	RAMP4:RAMP_INT;
	RAMP5:RAMP_INT;
	RAMP6:RAMP_INT;
	RAMP7:RAMP_INT;
	RAMP8:RAMP_INT;
	RAMP9:RAMP_INT;
	RAMP10:RAMP_INT;
	RAMP11:RAMP_INT;
	RAMP12:RAMP_INT;
	RAMP13:RAMP_INT;
	RAMP14:RAMP_INT;
	RAMP15:RAMP_INT;
	RAMP16:RAMP_INT;
	RAMP17:RAMP_INT;
	RAMP18:RAMP_INT;
	RAMP19:RAMP_INT;
	RAMP20:RAMP_INT;
	RAMP21:RAMP_INT;
	RAMP22:RAMP_INT;
	RAMP23:RAMP_INT;
	RAMP24:RAMP_INT;
	PWM_Y23_SET_Taget1:INT;
	PWM_Y24_SET_Taget1:INT;
	PWM_Y18_SET_Taget1:INT;
	PWM_Y18_SET_Taget:UINT;
	ASCEND_value2:INT;
	//2023 01 13 增加
	//行走动作斜坡值
	R_RAMP_traval:INT:=800;
	F_RAMP_traval:INT:=400;
	TIMEBASE_traval:TIME:=T#200MS;
	//动力头动作斜坡值
	R_RAMP_ratate:INT:=800;
	F_RAMP_ratate:INT:=800;
	TIMEBASE_ratate:TIME:=T#100MS;
	//主卷扬动作斜坡值
	R_RAMP_mainwinch:INT:=800;
	F_RAMP_mainwinch_up:INT:=400;
	F_RAMP_mainwinch_down:INT:=400;
	TIMEBASE_mainwinch:TIME:=T#200MS;
	//主泵排量斜坡值
	R_RAMP_pump:INT:=300;
	F_RAMP_pump:INT:=1000;
	TIMEBASE_pump:TIME:=T#1000MS;
	//卸荷阀斜坡值
	R_RAMP_xiehe:INT:=500;
	F_RAMP_xiehe:INT:=400;
	TIMEBASE_xiehe:TIME:=T#500MS;
	
	//直线阀斜坡值
	R_RAMP_zhixian:INT:=800;
	F_RAMP_zhixian:INT:=800;
	TIMEBASE_zhixian:TIME:=T#300MS;
		
	Subtract: BOOL;
	TIME_LvBo4:TON;
	Curve_input:UINT;
	Curve_Par: SINT:=0;
	Curve_Par1: SINT:=0;
	Move_JOY_FUHE: UINT;
	PWM_JOY_Jiao_L_UP1:UINT;
	PWM_JOY_Jiao_L_DOWN1:UINT;
	PWM_JOY_Jiao_R_UP1:UINT;
	PWM_JOY_Jiao_R_DOWN1:UINT;
	
	PWM_JOYX_R_UP_a:UINT;
	PWM_JOYX_R_UP_b:UINT;
	
	PWM_JOYX_R_DOWN_a:UINT;
	PWM_JOYX_R_DOWN_b:UINT;
	
	PWM_JOYY_L_DOWN_a:UINT;
	PWM_JOYY_L_DOWN_b:UINT;
	
	PWM_JOYY_L_UP_a:UINT;
	PWM_JOYY_L_UP_b:UINT;
	aaaa:UINT:=500;
	
	JOY_PAOTU:BOOL;
	
	JOY_PAOTU_tiaojian:BOOL;
	TIME_1000_1ms:ton;
	tempbool:BOOL;
	CANI_JOYX_R_last2:UINT;
	Sub_Joyx_r2:INT;
	JianGE11:REAL:=2;
	JianGE21:uint:=10;
	END_IFc: INT;
	x1:UINT:=8;
	x2:UINT:=8;
	PWM_JOY_JIAO:UINT;
	PWM_Y39_SET1:UINT;
	PWM_Y40_SET1:UINT;
	aaa: INT;
	TIME_50ms:TON;
	TIME_55ms:TOF;
	TIME_2000ms:TOF;
	start_move: BOOL;
	T1:TIME;
	TEMP1:UINT;
	X3: INT;
	X4: INT;
	liandong:BOOL;
	PWM_Y9_SET1:INT;
	PWM_Y10_SET1:INT;
	PWM_Y13_SET1:INT;
	PWM_Y14_SET1:INT;
	yanchi1:BOOL;
	yanchi_ton1:ton;
	RAMP15_IN:UINT;
	RAMP16_IN:UINT;
	Rtrig_d1:R_TRIG;
	Rtrig_d2:R_TRIG;
	
	Rtrig_DongLiTou1:R_TRIG;
	Rtrig_DongLiTou2:R_TRIG;
	Count_TIMES_Fanzhuan: UINT;
	Count_TIMES_Zhengzhuan: UINT;
	TIME_1000ms:TON;
	TIME_1000ms_TP:TON;
	Count_TIMES_Fanzhuan_LAST: UINT;
	Count_TIMES_Zhengzhuan_LAST: UINT;
	Paotu_Modle: BOOL;
	PaoTU_biaozhi: BOOL;
	TIMEBASE_D: TIME;
	PWM_Y39_SET_Target1:INT;
	PWM_Y40_SET_Target1:INT;
	PWM_Y37_SET_Target:UINT;
	PWM_Y17_SET2:UINT;
	t_PowerHead_move:TON;
	x_t_PowerHead_move:INT:=10;//100-10
	x2_t_PowerHead_move:INT:=10;//100-10
	P_value:REAL;//动力头反转+主卷上提时的分流系数
	PWM_JOY_P:UINT;
	PWM_JOY_P1:UINT;
	PWM_JOY_P2:UINT;
	PWM_JOY_P3:UINT;
	PWM_JOY_P4:UINT;
	ASCEND_value:INT;
	ftp1:INT:=500;
	ftp2:INT:=100;
	t_powertime:TIME;
	
	P25_Flag:BOOL;
	P27_Flag:BOOL;
	P29_Flag:BOOL;
	P31_Flag:BOOL;
	PressLvBo_TON:TON;
	PressLvBo_TON1: TON;
	PressLvBo_TON2: TON;
	PressLvBo_TON3: TON;
	test: BYTE;
	testpaotu: UINT := 450;
	Y33_2:UINT:=370;
	Y33_1:UINT:=200;
END_VAR

//动力头反转与主卷上提时的分流系数值
(*IF CANO_ZhuJuanPressure<=100 THEN
	P_value:=TO_REAL(PAR_KI+40)/100.0;
ELSIF CANO_ZhuJuanPressure>100 AND  CANO_ZhuJuanPressure<=200 THEN
	P_value:=TO_REAL(PAR_KI+20)/100.0;
ELSE
	P_value:=TO_REAL(PAR_KI)/100;
END_IF*)
P_value:=TO_REAL(PAR_KI)/100;  //出厂值设定为35
//喇叭
IF DI_LHandle_SB5 THEN
	DOH_Y59:=TRUE;
ELSE
	DOH_Y59:=FALSE;
END_IF
//延时断电
TIME_2000ms(IN:=DIH_power3,PT:=T#2S);
IF(TIME_2000ms.Q)THEN
	DOH_YS3:=TRUE;
ELSE
	DOH_YS3:=FALSE;
END_IF

//主卷上限位及解锁
IF(DI_LHandle_SB1 AND (NOT CANI_WorkModeSwitch))THEN
	JieSuoBool:=TRUE;
ELSE
	JieSuoBool:=FALSE;	
END_IF

IF DIL_SQ4 THEN
	IF(NOT JieSuoBool) THEN
		PWM_JOYY_L_DOWN:=0;
	END_IF
END_IF

//主卷下限位及解锁
//主卷下放限制
IF( CANO_MainWinchTension*100<PAR_MainWinchLaLi_Low) AND (NOT DI_LHandle_SB1) AND (CANI_WorkModeSwitch)THEN
	PWM_JOYY_L_UP:=0;
END_IF

TIME_50ms(in:=start_move,pt:=T1);
TIME_55ms(in:=start_move,pt:=T#500MS);
IF( LeftMove_move OR  RightMove_move  OR   MainWinch_move OR PowerHead_move OR ViceWinch_move )THEN
	start_move:=TRUE;
ELSE
	start_move:=FALSE;
END_IF
	 


IF NOT DIL_SQ3 THEN(*先导控制输入*)
	IF PWM_JOYX_L_UP>10 OR PWM_JOYX_L_DOWN>10 THEN  DI_PWM_JOYX_L := TRUE;ELSE DI_PWM_JOYX_L:=FALSE;END_IF(*左手柄左右动作*)
	IF PWM_JOYY_L_UP>10 OR PWM_JOYY_L_DOWN>10 THEN  DI_PWM_JOYY_L := TRUE;ELSE DI_PWM_JOYY_L:=FALSE;END_IF(*左手柄前后动作*)
	IF PWM_JOYX_R_UP>10 OR PWM_JOYX_R_DOWN>10 THEN  DI_PWM_JOYX_R := TRUE;ELSE DI_PWM_JOYX_R:=FALSE;END_IF(*右手柄左右动作*)
	IF PWM_JOYY_R_UP>10 OR PWM_JOYY_R_DOWN>10 THEN  DI_PWM_JOYY_R := TRUE;ELSE DI_PWM_JOYY_R:=FALSE;END_IF(*右手柄前后动作*)
	IF PWM_JOY_Jiao_L_UP>10 OR PWM_JOY_Jiao_L_DOWN>10 THEN  DI_PWM_JOY_Jiao_L:= TRUE;ELSE DI_PWM_JOY_Jiao_L:=FALSE;END_IF(*左脚踏前后动作*)
	IF PWM_JOY_Jiao_R_UP>10 OR PWM_JOY_Jiao_R_DOWN>10 THEN  DI_PWM_JOY_Jiao_R := TRUE;ELSE DI_PWM_JOY_Jiao_R:=FALSE;END_IF(*左脚踏左右动作*)
ELSE
	DI_PWM_JOYX_L:=FALSE;
	DI_PWM_JOYY_L:=FALSE;
	DI_PWM_JOYX_R:=FALSE;
	DI_PWM_JOYY_R:=FALSE;
	DI_PWM_JOY_Jiao_L:=FALSE;
	DI_PWM_JOY_Jiao_R:=FALSE;
END_IF

(*动作标志*)
IF DI_PWM_JOYY_L THEN MainWinch_move:=TRUE; ELSE MainWinch_move:=FALSE;END_IF(*主卷扬动作*)
IF DI_PWM_JOYX_L THEN Rotation_move:=TRUE; ELSE Rotation_move:=FALSE;END_IF(*回转动作*)
IF CANI_WorkModeSwitch THEN   (*作业挡情况下*)
	IF DI_PWM_JOYX_R THEN PowerHead_move:=TRUE;ELSE PowerHead_move:=FALSE;END_IF(*动力头回转动作*)
	IF DI_PWM_JOYY_R THEN JiaYa_move:=TRUE;ELSE JiaYa_move:=FALSE;END_IF(*动力头加压动作*)
	LvZhang_move:=FALSE;
	BianFu_move:=FALSE;
	ViceWinch_move:=FALSE;
	LeftMove_move:=FALSE;
	RightMove_move:=FALSE;
ELSE   (*调整档状态*)
	IF DI_PWM_JOYX_R THEN  LvZhang_move:=TRUE;ELSE LvZhang_move:=FALSE;END_IF(*L履带、张紧、支腿动作,M4阀*)
	(*LeftMove_move:=DI_PWM_JOY_Jiao_L;(*左行走动作*)
	RightMove_move:=DI_PWM_JOY_Jiao_R;*)(*右行走动作*)
	IF( PWM_JOY_Jiao_L_UP1>10 OR PWM_JOY_Jiao_L_DOWN1>10)  AND  DI_PWM_JOY_Jiao_L THEN
		LeftMove_move:=TRUE;
	ELSE
		LeftMove_move:=FALSE;
	END_IF
	IF( PWM_JOY_Jiao_R_UP1>10 OR PWM_JOY_Jiao_R_DOWN1>10)  AND  DI_PWM_JOY_Jiao_R THEN
		RightMove_move:=TRUE;
	ELSE
		RightMove_move:=FALSE;
	END_IF

	IF  DI_RHandle_SB5 THEN
		ViceWinch_move:=FALSE;
		IF  DI_PWM_JOYY_R  THEN BianFu_move:=TRUE;ELSE BianFu_move:=FALSE;END_IF(*变幅动作M4阀*)
	ELSE
		BianFu_move:=FALSE;
		IF DI_PWM_JOYY_R  THEN ViceWinch_move:=TRUE;ELSE ViceWinch_move:=FALSE;END_IF(*副卷扬动作M4阀*)
	END_IF
	PowerHead_move:=FALSE;
	JiaYa_move:=FALSE;
END_IF


(****主阀单动作标志****)
	IF (NOT MainWinch_move) AND (NOT PowerHead_move) AND (ViceWinch_move) THEN
		Single_move:=TRUE;
	ELSE
		Single_move:=FALSE;
	END_IF
	
//先导控制
IF(NOT DIL_SQ3) AND NOT VarGpsSystemLockedState THEN
	DOH_Y51:=TRUE;
ELSE
	DOH_Y51:=FALSE;
END_IF

//行走动作
(*脚踏阀偏差*)
IF   ((PWM_JOY_Jiao_L_UP-PWM_JOY_Jiao_R_UP)<200 OR(PWM_JOY_Jiao_R_UP-PWM_JOY_Jiao_L_UP)<200) THEN
	PWM_JOY_Jiao_L_UP1:=MAX(PWM_JOY_Jiao_L_UP,PWM_JOY_Jiao_R_UP);
	PWM_JOY_Jiao_R_UP1:=MAX(PWM_JOY_Jiao_L_UP,PWM_JOY_Jiao_R_UP);
ELSE
	PWM_JOY_Jiao_L_UP1:=PWM_JOY_Jiao_L_UP;
	PWM_JOY_Jiao_R_UP1:=PWM_JOY_Jiao_R_UP;
END_IF
IF   ((PWM_JOY_Jiao_L_DOWN-PWM_JOY_Jiao_R_DOWN)<200  OR  (PWM_JOY_Jiao_R_DOWN-PWM_JOY_Jiao_L_DOWN)<200 ) THEN
	PWM_JOY_Jiao_L_DOWN1:=MAX(PWM_JOY_Jiao_L_DOWN,PWM_JOY_Jiao_R_DOWN);
	PWM_JOY_Jiao_R_DOWN1:=MAX(PWM_JOY_Jiao_L_DOWN,PWM_JOY_Jiao_R_DOWN);
ELSE
	PWM_JOY_Jiao_L_DOWN1:=PWM_JOY_Jiao_L_DOWN;
	PWM_JOY_Jiao_R_DOWN1:=PWM_JOY_Jiao_R_DOWN;
END_IF

PWM_JOY_JIAO:=MAX(PWM_JOY_Jiao_L_UP1,PWM_JOY_Jiao_R_UP1,PWM_JOY_Jiao_L_DOWN1,PWM_JOY_Jiao_R_DOWN1);
liandong:=FALSE;
(*左行走*)
(*泵1   Y1   Y39控制右行走   Y15  16 *)
(*泵2   Y2 Y40 控制左行走    Y5  Y6*)
IF LeftMove_move THEN
	IF PWM_JOY_Jiao_L_UP1>10 THEN
		PWM_Y2_Target:=REAL_TO_UINT(UINT_TO_REAL(PWM_JOY_Jiao_L_UP1)/1000*(PAR_Y1_1_PosFull-PAR_Y1_1_NegFull)+PAR_Y1_1_NegFull);
		PWM_Y5_SET_Target:=REAL_TO_UINT(UINT_TO_REAL(PWM_JOY_Jiao_L_UP1)/1000*(PAR_Valve2_PosFull-PAR_Valve2_NegFull)+PAR_Valve2_NegFull);
		PWM_Y6_SET_Target:=0;	
	ELSIF PWM_JOY_Jiao_L_DOWN1>10 THEN
		PWM_Y2_Target:=REAL_TO_UINT(UINT_TO_REAL(PWM_JOY_Jiao_L_DOWN1)/1000*(PAR_Y1_1_PosFull-PAR_Y1_1_NegFull)+PAR_Y1_1_NegFull);
		PWM_Y6_SET_Target:=REAL_TO_UINT(UINT_TO_REAL(PWM_JOY_Jiao_L_DOWN1)/1000*(PAR_Valve2_PosFull-PAR_Valve2_NegFull)+PAR_Valve2_NegFull);
		PWM_Y5_SET_Target:=0;		
	END_IF
ELSE
	PWM_Y5_SET_Target:=0;
	PWM_Y6_SET_Target:=0;
END_IF
(*右行走*)
IF RightMove_move  THEN
	IF PWM_JOY_Jiao_R_UP1>10 THEN
		PWM_Y1_Target:=REAL_TO_UINT(UINT_TO_REAL(PWM_JOY_Jiao_R_UP1)/1000*(PAR_Y1_1_PosFull-PAR_Y1_1_NegFull)+PAR_Y1_1_NegFull);
		PWM_Y15_SET_Target:=REAL_TO_UINT(UINT_TO_REAL(PWM_JOY_Jiao_R_UP1)/1000*(PAR_Valve1_PosFull-PAR_Valve1_NegFull)+PAR_Valve1_NegFull);
		PWM_Y16_SET_Target:=0;
	
	ELSIF PWM_JOY_Jiao_R_DOWN1>10 THEN
		PWM_Y1_Target:=REAL_TO_UINT(UINT_TO_REAL(PWM_JOY_Jiao_R_DOWN1)/1000*(PAR_Y1_1_PosFull-PAR_Y1_1_NegFull)+PAR_Y1_1_NegFull);
		PWM_Y16_SET_Target:=REAL_TO_UINT(UINT_TO_REAL(PWM_JOY_Jiao_R_DOWN1)/1000*(PAR_Valve1_PosFull-PAR_Valve1_NegFull)+PAR_Valve1_NegFull);
		PWM_Y15_SET_Target:=0;
		
	END_IF
ELSE
	PWM_Y15_SET_Target:=0;
	PWM_Y16_SET_Target:=0;
END_IF

	//如有必要，可根据行走阀开关大小调整斜坡值
(*	IF(PWM_Y5_SET<1000  AND  PWM_Y5_SET>=900)THEN
			R_RAMP_traval:=100;
	ELSIF(PWM_Y5_SET<900 AND PWM_Y5_SET>=780)THEN
			R_RAMP_traval:=10;
	ELSE
			R_RAMP_traval:=250;
	END_IF
		
	IF(PWM_Y6_SET<1000  AND  PWM_Y6_SET>=900)THEN
			F_RAMP_traval:=100;		
	ELSIF(PWM_Y6_SET<900 AND PWM_Y6_SET>750 )THEN
			F_RAMP_traval:=15;
	ELSE
			F_RAMP_traval:=250;
	END_IF*)
	
(*行走动作缓冲*)
RAMP11(
	IN:=WORD_TO_INT(PWM_Y5_SET_Target), 
	ASCEND:= R_RAMP_traval, 
	DESCEND:= F_RAMP_traval, 
	TIMEBASE:=TIMEBASE_traval , 
	RESET:=FALSE , 
	OUT=>(PWM_Y5_SET_Target1));
IF(PWM_Y5_SET_Target1>=400) THEN
	Curve_input:=TO_UINT(PWM_Y5_SET_Target1 - 400);
	IF(Curve_input>900) THEN
		Curve_input:=900;
	END_IF
	curve11(input:=REAL_TO_UINT(UINT_TO_REAL(Curve_input)*72.8),Zero:=FALSE,Full:=FALSE,
		   PAR_Progression:=Curve_Par1,OutputEnable:=TRUE);
	PWM_Y5_SET:=PAR_Valve1_NegFull + REAL_TO_UINT(UINT_TO_REAL(curve11.Output)/72.8);
ELSE
	PWM_Y5_SET:=0;
END_IF

RAMP12(
	IN:=WORD_TO_INT(PWM_Y6_SET_Target), 
	ASCEND:= R_RAMP_traval, 
	DESCEND:= F_RAMP_traval, 
	TIMEBASE:=TIMEBASE_traval , 
	RESET:=FALSE , 
	OUT=>(PWM_Y6_SET_Target1));
IF(PWM_Y6_SET_Target1>=400) THEN
	Curve_input:=TO_UINT(PWM_Y6_SET_Target1 - 400);
	IF(Curve_input>900) THEN
		Curve_input:=900;
	END_IF
	curve12(input:=REAL_TO_UINT(UINT_TO_REAL(Curve_input)*72.8),Zero:=FALSE,Full:=FALSE,
		   PAR_Progression:=Curve_Par1,OutputEnable:=TRUE);
	PWM_Y6_SET:=PAR_Valve1_NegFull + REAL_TO_UINT(UINT_TO_REAL(curve12.Output)/72.8);
ELSE
	PWM_Y6_SET:=0;
END_IF

RAMP13(
	IN:=WORD_TO_INT(PWM_Y15_SET_Target), 
	ASCEND:= R_RAMP_traval, 
	DESCEND:= F_RAMP_traval, 
	TIMEBASE:=TIMEBASE_traval , 
	RESET:=FALSE , 
	OUT=>(PWM_Y15_SET_Target1));
IF(PWM_Y15_SET_Target1>=400) THEN
	Curve_input:=TO_UINT(PWM_Y15_SET_Target1 - 400);
	IF(Curve_input>900) THEN
		Curve_input:=900;
	END_IF
	curve13(input:=REAL_TO_UINT(UINT_TO_REAL(Curve_input)*72.8),Zero:=FALSE,Full:=FALSE,
		   PAR_Progression:=Curve_Par1,OutputEnable:=TRUE);
	PWM_Y15_SET:=PAR_Valve1_NegFull + REAL_TO_UINT(UINT_TO_REAL(curve13.Output)/72.8);
ELSE
	PWM_Y15_SET:=0;
END_IF

RAMP14(
	IN:=WORD_TO_INT(PWM_Y16_SET_Target), 
	ASCEND:= R_RAMP_traval, 
	DESCEND:= F_RAMP_traval, 
	TIMEBASE:=TIMEBASE_traval , 
	RESET:=FALSE , 
	OUT=>(PWM_Y16_SET_Target1));
IF(PWM_Y16_SET_Target1>=400) THEN
	Curve_input:=TO_UINT(PWM_Y16_SET_Target1 - 400);
	IF(Curve_input>900) THEN
		Curve_input:=900;
	END_IF
	curve14(input:=REAL_TO_UINT(UINT_TO_REAL(Curve_input)*72.8),Zero:=FALSE,Full:=FALSE,
		   PAR_Progression:=Curve_Par1,OutputEnable:=TRUE);
	PWM_Y16_SET:=PAR_Valve1_NegFull + REAL_TO_UINT(UINT_TO_REAL(curve14.Output)/72.8);
ELSE
	PWM_Y16_SET:=0;
END_IF


(*直线行走*)
(*IF(  DIH_SA19)THEN
	IF (PWM_JOY_Jiao_L_UP1>10  AND PWM_JOY_Jiao_R_UP1>10) OR ( PWM_JOY_Jiao_L_DOWN1>10 AND PWM_JOY_Jiao_R_DOWN1>10)THEN
		PWM_Y37_SET_Target:=800;  //开环  占控比   0-1000
	ELSE
		PWM_Y37_SET_Target:=0;
	END_IF
ELSE
	PWM_Y37_SET_Target:=0;
END_IF

IF((LeftMove_move OR RightMove_move)AND MainWinch_move)THEN
	PWM_Y1_Target:=REAL_TO_UINT(UINT_TO_REAL(PWM_JOY_JIAO)/1000*(PAR_Y2_PosFull-PAR_Y2_NegFull)+PAR_Y2_NegFull);
	PWM_Y2_Target:=0;
	PWM_Y37_SET_Target:=800;
END_IF*)
(*直线行走*)//Y2  Y40   行走阀
IF DIH_SA19 THEN
	PWM_Y37_SET_Target:=800;
	PWM_Y1_Target:=0;
ELSE
	PWM_Y37_SET_Target:=0;
END_IF

IF((LeftMove_move OR RightMove_move)AND MainWinch_move)THEN
	PWM_Y2_Target:=REAL_TO_UINT(UINT_TO_REAL(PWM_JOY_JIAO)/1000*(PAR_Y2_PosFull-PAR_Y2_NegFull)+PAR_Y2_NegFull);
	PWM_Y1_Target:=0;
	PWM_Y37_SET_Target:=800;
END_IF


RAMP21(
	IN:=UINT_TO_INT(PWM_Y37_SET_Target), 
	ASCEND:= R_RAMP_zhixian, 
	DESCEND:= F_RAMP_zhixian, 
	TIMEBASE:=TIMEBASE_zhixian , 
	RESET:=FALSE , 
	OUT=>(PWM_Y37_SET));


IF(PWM_JOYX_R_UP<=500)THEN
	PWM_JOYX_R_UP_a:=PWM_JOYX_R_UP;
	PWM_JOYX_R_UP_b:=0;
ELSE
	PWM_JOYX_R_UP_a:=500;
	PWM_JOYX_R_UP_b:=PWM_JOYX_R_UP-500;
END_IF

IF(PWM_JOYX_R_DOWN<=500)THEN
	PWM_JOYX_R_DOWN_a:=PWM_JOYX_R_DOWN;
	PWM_JOYX_R_DOWN_b:=0;
ELSE
	PWM_JOYX_R_DOWN_a:=500;
	PWM_JOYX_R_DOWN_b:=PWM_JOYX_R_DOWN-500;
END_IF

	
(*单动力头动作*)
IF (NOT MainWinch_move) AND(PowerHead_move) AND(NOT DI_RHandle_SB6) THEN
	IF PWM_JOYX_R_UP>10 THEN//动力头反转
			PWM_Y1_Target:=REAL_TO_UINT(UINT_TO_REAL(PWM_JOYX_R_UP)/1000*(PAR_Y1_PosFull-PAR_Y1_NegFull)+PAR_Y1_NegFull);			
			PWM_Y2_Target:=REAL_TO_UINT(UINT_TO_REAL(PWM_JOYX_R_UP_b)/500*(PAR_Y2_PosFull-PAR_Y2_NegFull)+PAR_Y2_NegFull);
		IF(DIH_SA18)THEN
			PWM_Y1_Target:=0;			
			PWM_Y2_Target:=REAL_TO_UINT(UINT_TO_REAL(PWM_JOYX_R_UP)/1000*(PAR_Y2_PosFull-PAR_Y2_NegFull)+PAR_Y2_NegFull);
		END_IF
		PWM_Y12_SET_Tatget:=REAL_TO_UINT(UINT_TO_REAL(PWM_JOYX_R_UP)/1000*(PAR_Valve1_PosFull-PAR_Valve1_NegFull)+PAR_Valve1_NegFull);
		PWM_Y61_SET_Tatget:=REAL_TO_UINT(UINT_TO_REAL(PWM_JOYX_R_UP)/1000*(PAR_Valve1_PosFull-PAR_Valve1_NegFull)+PAR_Valve1_NegFull);
		PWM_Y14_SET_Tatget:=REAL_TO_UINT(UINT_TO_REAL(PWM_JOYX_R_UP_b)/500*(PAR_Valve2_PosFull-PAR_Valve2_NegFull)+PAR_Valve2_NegFull);
		PWM_Y11_SET:=0;
		PWM_Y13_SET:=0;
		PWM_Y60_SET:=0;
		PWM_Y11_SET_Tatget:=0;
		PWM_Y13_SET_Tatget:=0;
		PWM_Y60_SET_Tatget:=0;
		IF(PWM_JOYX_R_UP>700)THEN
			PWM_Y41_SET:=PAR_Valve2_PosFull;//快速回油阀
		END_IF
		PWM_Y59_SET:=0;
		PWM_Y42_SET:=0;
	ELSIF PWM_JOYX_R_DOWN>10 THEN //动力头正转
			PWM_Y1_Target:=REAL_TO_UINT(UINT_TO_REAL(PWM_JOYX_R_DOWN)/1000*(PAR_Y1_PosFull-PAR_Y1_NegFull)+PAR_Y1_NegFull);			
			PWM_Y2_Target:=REAL_TO_UINT(UINT_TO_REAL(PWM_JOYX_R_DOWN_b)/500*(PAR_Y2_PosFull-PAR_Y2_NegFull)+PAR_Y2_NegFull);
		IF(DIH_SA18)THEN
			PWM_Y1_Target:=0;			
			PWM_Y2_Target:=REAL_TO_UINT(UINT_TO_REAL(PWM_JOYX_R_DOWN)/1000*(PAR_Y2_PosFull-PAR_Y2_NegFull)+PAR_Y2_NegFull);
		END_IF
			PWM_Y11_SET_Tatget:=REAL_TO_UINT(UINT_TO_REAL(PWM_JOYX_R_DOWN)/1000*(PAR_Valve1_PosFull-PAR_Valve1_NegFull)+PAR_Valve1_NegFull);
			PWM_Y60_SET_Tatget:=REAL_TO_UINT(UINT_TO_REAL(PWM_JOYX_R_DOWN)/1000*(PAR_Valve1_PosFull-PAR_Valve1_NegFull)+PAR_Valve1_NegFull);		
			PWM_Y13_SET_Tatget:=REAL_TO_UINT(UINT_TO_REAL(PWM_JOYX_R_DOWN_b)/500*(PAR_Valve2_PosFull-PAR_Valve2_NegFull)+PAR_Valve2_NegFull);
		IF(PWM_JOYX_R_DOWN>700)THEN
		PWM_Y59_SET:=PAR_Valve2_PosFull;//合流
		PWM_Y42_SET:=PAR_Valve2_PosFull;//快速回油阀
		END_IF
		PWM_Y41_SET:=0;
		PWM_Y12_SET:=0;
		PWM_Y14_SET:=0;
		PWM_Y61_SET:=0;	
		PWM_Y12_SET_Tatget:=0;
		PWM_Y14_SET_Tatget:=0;
		PWM_Y61_SET_Tatget:=0;
	END_IF
ELSIF (MainWinch_move) AND(PowerHead_move) AND( NOT DI_RHandle_SB6) THEN
	//主卷和动力头复合动作时 主泵2提供给动力头油
	IF PWM_JOYX_R_UP>10 THEN//动力头反转 
		IF(PWM_JOYY_L_DOWN>10) THEN//主卷上提
		PWM_JOY_P:=MAX(PWM_JOYY_L_DOWN,PWM_JOYX_R_UP);
		PWM_Y1_Target:=REAL_TO_UINT(UINT_TO_REAL(PWM_JOY_P)/1000*(PAR_Y2_PosFull-PAR_Y2_NegFull)+PAR_Y2_NegFull);
		PWM_Y12_SET_Tatget:=REAL_TO_UINT(UINT_TO_REAL(PWM_JOYX_R_UP)/1000*(PAR_Valve2_PosFull-400)*P_value+400);
		PWM_Y11_SET_Tatget:=0;
		PWM_Y14_SET_Tatget:=0;
		PWM_Y13_SET_Tatget:=0;
		PWM_Y60_SET_Tatget:=0;
		PWM_Y61_SET_Tatget:=0;
		PWM_Y41_SET:=PAR_Valve2_PosFull;
		PWM_Y42_SET:=0;
		PWM_Y59_SET:=0;
		ELSIF PWM_JOYY_L_UP>10 THEN//主卷下放
 		PWM_Y1_Target:=REAL_TO_UINT(UINT_TO_REAL(PWM_JOYX_R_UP)/1000*(PAR_Y2_PosFull-PAR_Y2_NegFull)+PAR_Y2_NegFull);
		PWM_Y12_SET_Tatget:=REAL_TO_UINT(UINT_TO_REAL(PWM_JOYX_R_UP)/1000*(PAR_Valve2_PosFull-PAR_Valve2_NegFull)+PAR_Valve2_NegFull);
		PWM_Y11_SET_Tatget:=0;
		PWM_Y14_SET_Tatget:=0;
		PWM_Y13_SET_Tatget:=0;
		PWM_Y60_SET_Tatget:=0;
		PWM_Y61_SET_Tatget:=0;
		PWM_Y41_SET:=PAR_Valve2_PosFull;
		PWM_Y59_SET:=0;	
		PWM_Y42_SET:=0;
		END_IF
		
		
	ELSIF PWM_JOYX_R_DOWN>10 THEN //动力头正转
		PWM_Y1_Target:=REAL_TO_UINT(UINT_TO_REAL(PWM_JOYX_R_DOWN)/1000*(PAR_Y2_PosFull-PAR_Y2_NegFull)+PAR_Y2_NegFull);
		PWM_Y11_SET_Tatget:=REAL_TO_UINT(UINT_TO_REAL(PWM_JOYX_R_DOWN)/1000*(PAR_Valve2_PosFull-PAR_Valve2_NegFull)+PAR_Valve2_NegFull);
		PWM_Y13_SET_Tatget:=0;
		PWM_Y12_SET_Tatget:=0;
		PWM_Y14_SET_Tatget:=0;
		PWM_Y60_SET_Tatget:=0;
		PWM_Y61_SET_Tatget:=0;
		PWM_Y41_SET:=0;
		PWM_Y42_SET:=PAR_Valve2_PosFull;
		PWM_Y59_SET:=0;	
	END_IF	
ELSE
		PWM_Y12_SET_Tatget:=0;
		PWM_Y14_SET_Tatget:=0;
		PWM_Y61_SET_Tatget:=0;
		PWM_Y11_SET_Tatget:=0;
		PWM_Y13_SET_Tatget:=0;
		PWM_Y60_SET_Tatget:=0;
		PWM_Y41_SET:=0;
		PWM_Y42_SET:=0;	
		PWM_Y59_SET:=0;	
END_IF


//判断抛土模式
Rtrig_DongLiTou1(clk:=(CANI_JOYX_R>3000));//反转判断
IF Rtrig_DongLiTou1.Q THEN
	Count_TIMES_Fanzhuan:=Count_TIMES_Fanzhuan + 1;
END_IF
Rtrig_DongLiTou2(clk:=(CANI_JOYX_R<2000));//正转判断
IF Rtrig_DongLiTou2.Q THEN
	Count_TIMES_Zhengzhuan:=Count_TIMES_Zhengzhuan + 1;
END_IF	
IF (Count_TIMES_Fanzhuan_LAST<>Count_TIMES_Fanzhuan) AND (Count_TIMES_Zhengzhuan_LAST<>Count_TIMES_Zhengzhuan) THEN
	Paotu_Modle:=TRUE;
END_IF
TIME_1000ms(IN:=NOT TIME_1000ms.Q,PT:=T#800MS);
IF (TIME_1000ms.Q) THEN
	Count_TIMES_Fanzhuan_LAST:=Count_TIMES_Fanzhuan;
	Count_TIMES_Zhengzhuan_LAST:=Count_TIMES_Zhengzhuan;
END_IF

IF(Count_TIMES_Fanzhuan_LAST=Count_TIMES_Fanzhuan) AND (Count_TIMES_Zhengzhuan_LAST=Count_TIMES_Zhengzhuan) THEN
	PaoTU_biaozhi:=TRUE;
ELSE
	PaoTU_biaozhi:=FALSE;	
END_IF
TIME_1000ms_TP(IN:=PaoTU_biaozhi,PT:=T#800MS);
IF TIME_1000ms_TP.Q OR MainWinch_move  THEN
	Paotu_Modle:=FALSE;
END_IF

IF(NOT CANI_WorkModeSwitch) THEN
	Paotu_Modle:=FALSE;
END_IF

IF Paotu_Modle THEN
	TIMEBASE_ratate:=T#20MS;
ELSE
	TIMEBASE_ratate:=T#100MS;
END_IF


(*动力头动作缓冲*)
//启动缓冲时间300ms，停止缓冲时间600ms
(*动力头动作缓冲*)
//启动缓冲时间300ms，停止缓冲时间600ms
RAMP1(
	IN:=WORD_TO_INT(PWM_Y11_SET_Tatget), 
	ASCEND:= R_RAMP_ratate, 
	DESCEND:= F_RAMP_ratate, 
	TIMEBASE:=TIMEBASE_ratate , 
	RESET:=FALSE , 
	OUT=>(PWM_Y11_SET_Tatget1));
IF(PWM_Y11_SET_Tatget1>=400) THEN
	Curve_input:=TO_UINT(PWM_Y11_SET_Tatget1 - 400);
	IF(Curve_input>900) THEN
		Curve_input:=900;
	END_IF
	curve1(input:=REAL_TO_UINT(UINT_TO_REAL(Curve_input)*72.8),Zero:=FALSE,Full:=FALSE,
		   PAR_Progression:=Curve_Par,OutputEnable:=TRUE);
	PWM_Y11_SET:=PAR_Valve1_NegFull + REAL_TO_UINT(UINT_TO_REAL(curve1.Output)/72.8);
ELSE
	PWM_Y11_SET:=0;
END_IF

RAMP2(
	IN:=WORD_TO_INT(PWM_Y12_SET_Tatget), 
	ASCEND:= R_RAMP_ratate, 
	DESCEND:= F_RAMP_ratate, 
	TIMEBASE:=TIMEBASE_ratate , 
	RESET:=FALSE , 
	OUT=>(PWM_Y12_SET_Tatget1));
IF(PWM_Y12_SET_Tatget1>=400) THEN
	Curve_input:=TO_UINT(PWM_Y12_SET_Tatget1 - 400);
	IF(Curve_input>900) THEN
		Curve_input:=900;
	END_IF
	curve2(input:=REAL_TO_UINT(UINT_TO_REAL(Curve_input)*72.8),Zero:=FALSE,Full:=FALSE,
		   PAR_Progression:=Curve_Par,OutputEnable:=TRUE);
	PWM_Y12_SET:=PAR_Valve1_NegFull + REAL_TO_UINT(UINT_TO_REAL(curve2.Output)/72.8);
ELSE
	PWM_Y12_SET:=0;
END_IF

RAMP3(
	IN:=WORD_TO_INT(PWM_Y13_SET_Tatget), 
	ASCEND:= R_RAMP_ratate, 
	DESCEND:= F_RAMP_ratate, 
	TIMEBASE:=TIMEBASE_ratate , 
	RESET:=FALSE , 
	OUT=>(PWM_Y13_SET_Tatget1));
IF(PWM_Y13_SET_Tatget1>=400) THEN
	Curve_input:=TO_UINT(PWM_Y13_SET_Tatget1 - 400);
	IF(Curve_input>900) THEN
		Curve_input:=900;
	END_IF
	curve3(input:=REAL_TO_UINT(UINT_TO_REAL(Curve_input)*72.8),Zero:=FALSE,Full:=FALSE,
		   PAR_Progression:=Curve_Par,OutputEnable:=TRUE);
	PWM_Y13_SET:=PAR_Valve1_NegFull + REAL_TO_UINT(UINT_TO_REAL(curve3.Output)/72.8);
ELSE
	PWM_Y13_SET:=0;
END_IF

RAMP4(
	IN:=WORD_TO_INT(PWM_Y14_SET_Tatget), 
	ASCEND:= R_RAMP_ratate, 
	DESCEND:= F_RAMP_ratate, 
	TIMEBASE:=TIMEBASE_ratate , 
	RESET:=FALSE , 
	OUT=>(PWM_Y14_SET_Tatget1));
IF(PWM_Y14_SET_Tatget1>=400) THEN
	Curve_input:=TO_UINT(PWM_Y14_SET_Tatget1 - 400);
	IF(Curve_input>900) THEN
		Curve_input:=900;
	END_IF
	curve4(input:=REAL_TO_UINT(UINT_TO_REAL(Curve_input)*72.8),Zero:=FALSE,Full:=FALSE,
		   PAR_Progression:=Curve_Par,OutputEnable:=TRUE);
	PWM_Y14_SET:=PAR_Valve1_NegFull + REAL_TO_UINT(UINT_TO_REAL(curve4.Output)/72.8);
ELSE
	PWM_Y14_SET:=0;
END_IF

RAMP5(
	IN:=WORD_TO_INT(PWM_Y60_SET_Tatget), 
	ASCEND:= R_RAMP_ratate, 
	DESCEND:= F_RAMP_ratate, 
	TIMEBASE:=TIMEBASE_ratate , 
	RESET:=FALSE , 
	OUT=>(PWM_Y60_SET_Tatget1));
IF(PWM_Y60_SET_Tatget1>=400) THEN
	Curve_input:=TO_UINT(PWM_Y60_SET_Tatget1 - 400);
	IF(Curve_input>900) THEN
		Curve_input:=900;
	END_IF
	curve5(input:=REAL_TO_UINT(UINT_TO_REAL(Curve_input)*72.8),Zero:=FALSE,Full:=FALSE,
		   PAR_Progression:=Curve_Par,OutputEnable:=TRUE);
	PWM_Y60_SET:=PAR_Valve1_NegFull + REAL_TO_UINT(UINT_TO_REAL(curve5.Output)/72.8);
ELSE
	PWM_Y60_SET:=0;
END_IF

RAMP6(
	IN:=WORD_TO_INT(PWM_Y61_SET_Tatget), 
	ASCEND:= R_RAMP_ratate, 
	DESCEND:= F_RAMP_ratate, 
	TIMEBASE:=TIMEBASE_ratate , 
	RESET:=FALSE , 
	OUT=>(PWM_Y61_SET_Tatget1));
IF(PWM_Y61_SET_Tatget1>=400) THEN
	Curve_input:=TO_UINT(PWM_Y61_SET_Tatget1 - 400);
	IF(Curve_input>900) THEN
		Curve_input:=900;
	END_IF
	curve6(input:=REAL_TO_UINT(UINT_TO_REAL(Curve_input)*72.8),Zero:=FALSE,Full:=FALSE,
		   PAR_Progression:=Curve_Par,OutputEnable:=TRUE);
	PWM_Y61_SET:=PAR_Valve1_NegFull + REAL_TO_UINT(UINT_TO_REAL(curve6.Output)/72.8);
ELSE
	PWM_Y61_SET:=0;
END_IF


IF(PWM_Y5_SET>1300)THEN
	PWM_Y5_SET :=1300;
END_IF
IF(PWM_Y6_SET>1300)THEN
	PWM_Y6_SET :=1300;
END_IF
IF(PWM_Y15_SET>1300)THEN
	PWM_Y15_SET :=1300;
END_IF
IF(PWM_Y16_SET>1300)THEN
	PWM_Y16_SET :=1300;
END_IF	
IF(PWM_Y11_SET>1300)THEN
	PWM_Y11_SET :=1300;
END_IF
IF(PWM_Y12_SET>1300)THEN
	PWM_Y12_SET :=1300;
END_IF
IF(PWM_Y13_SET>1300)THEN
	PWM_Y13_SET :=1300;
END_IF
IF(PWM_Y14_SET>1300)THEN
	PWM_Y14_SET :=1300;
END_IF
IF(PWM_Y60_SET>1300)THEN
	PWM_Y60_SET :=1300;
END_IF
IF(PWM_Y61_SET>1300)THEN
	PWM_Y61_SET :=1300;
END_IF


IF(PWM_Y11_SET<=300)THEN
	PWM_Y11_SET :=0;
END_IF
IF(PWM_Y12_SET<=300)THEN
	PWM_Y12_SET :=0;
END_IF
IF(PWM_Y13_SET<=300)THEN
	PWM_Y13_SET :=0;
END_IF
IF(PWM_Y14_SET<=300)THEN
	PWM_Y14_SET :=0;
END_IF
IF(PWM_Y60_SET<=300)THEN
	PWM_Y60_SET :=0;
END_IF
IF(PWM_Y61_SET<=300)THEN
	PWM_Y61_SET :=0;
END_IF


BiaoZHI_MainWinchUp:=FALSE;
IF(PWM_JOYY_L_UP<=500)THEN
	PWM_JOYY_L_UP_a:=PWM_JOYY_L_UP;
	PWM_JOYY_L_UP_b:=0;
ELSE
	PWM_JOYY_L_UP_a:=500;
	PWM_JOYY_L_UP_b:=PWM_JOYY_L_UP-500;
END_IF

IF(PWM_JOYY_L_DOWN<=500)THEN
	PWM_JOYY_L_DOWN_a:=PWM_JOYY_L_DOWN;
	PWM_JOYY_L_DOWN_b:=0;
ELSE
	PWM_JOYY_L_DOWN_a:=500;
	PWM_JOYY_L_DOWN_b:=PWM_JOYY_L_DOWN-500;
END_IF



(*单主卷动作*)
IF ( MainWinch_move) AND (NOT PowerHead_move) AND (NOT LeftMove_move) AND (NOT RightMove_move)THEN
	IF PWM_JOYY_L_UP>10   THEN//主卷下放
		PWM_Y1_Target:=REAL_TO_UINT(UINT_TO_REAL(PWM_JOYY_L_UP)/1000*(PAR_Y1_PosFull-PAR_Y1_NegFull)+PAR_Y1_NegFull);
		PWM_Y2_Target:=REAL_TO_UINT(UINT_TO_REAL(PWM_JOYY_L_UP)/1000*(PAR_Y2_PosFull-PAR_Y2_NegFull)+PAR_Y2_NegFull);
		BiaoZHI_MainWinchUp:=TRUE;
		PWM_Y8_SET_Target:=REAL_TO_UINT(UINT_TO_REAL(PWM_JOYY_L_UP)/1000*(PAR_Valve1_PosFull-PAR_Valve1_NegFull)+PAR_Valve1_NegFull);
		PWM_Y10_SET_Target:=REAL_TO_UINT(UINT_TO_REAL(PWM_JOYY_L_UP)/1000*(PAR_Valve2_PosFull-PAR_Valve2_NegFull)+PAR_Valve2_NegFull);
		PWM_Y7_SET_Target:=0;
		PWM_Y9_SET_Target:=0;
		IF(DIH_SA19)THEN
			PWM_Y10_SET_Target:=0;
			PWM_Y9_SET_Target:=0;
			PWM_Y2_Target:=0;	
		END_IF
	ELSIF PWM_JOYY_L_DOWN>10 THEN//主卷上提
		PWM_Y1_Target:=REAL_TO_UINT(UINT_TO_REAL(PWM_JOYY_L_DOWN)/1000*(PAR_Y1_PosFull-PAR_Y1_NegFull)+PAR_Y1_NegFull);
		PWM_Y2_Target:=REAL_TO_UINT(UINT_TO_REAL(PWM_JOYY_L_DOWN)/1000*(PAR_Y2_PosFull-PAR_Y2_NegFull)+PAR_Y2_NegFull);
		PWM_Y7_SET_Target:=REAL_TO_UINT(UINT_TO_REAL(PWM_JOYY_L_DOWN)/1000*(PAR_Valve1_PosFull-PAR_Valve2_NegFull)+PAR_Valve2_NegFull);
		PWM_Y9_SET_Target:=REAL_TO_UINT(UINT_TO_REAL(PWM_JOYY_L_DOWN)/1000*(PAR_Valve2_PosFull-PAR_Valve2_NegFull)+PAR_Valve2_NegFull);
		PWM_Y8_SET_Target:=0;
		PWM_Y10_SET_Target:=0;	
		IF(DIH_SA19)THEN
			PWM_Y10_SET_Target:=0;
			PWM_Y9_SET_Target:=0;
			PWM_Y2_Target:=0;	
		END_IF
	END_IF
ELSIF( MainWinch_move) AND (PowerHead_move) THEN
	//主卷和动力头复合动作时 主泵1提供给主卷油
	IF PWM_JOYY_L_UP>10 THEN//主卷下放
		IF(PWM_JOYX_R_DOWN>10) THEN //动力头正转
			PWM_JOY_P4:=MAX(PWM_JOYY_L_UP,PWM_JOYX_R_DOWN);
			PWM_Y2_Target:=REAL_TO_UINT(UINT_TO_REAL(PWM_JOYY_L_UP)/1000*(PAR_Y1_PosFull-PAR_Y1_NegFull)+PAR_Y1_NegFull);
			PWM_Y1_Target:=REAL_TO_UINT(UINT_TO_REAL(PWM_JOYY_L_UP)/1000*(PAR_Y1_PosFull-PAR_Y1_NegFull)+PAR_Y1_NegFull);
			PWM_Y10_SET_Target:=REAL_TO_UINT(UINT_TO_REAL(PWM_JOYY_L_UP)/1000*(PAR_Valve1_PosFull-PAR_Valve1_NegFull)+PAR_Valve1_NegFull);
			PWM_Y8_SET_Target:=REAL_TO_UINT(UINT_TO_REAL(1000-PWM_JOYX_R_DOWN)/1000*(PAR_Valve1_PosFull-PAR_Valve1_NegFull)+PAR_Valve1_NegFull);
			PWM_Y7_SET_Target:=0;
			PWM_Y9_SET_Target:=0;
		ELSIF PWM_JOYX_R_UP>10 THEN//动力头反转
			PWM_JOY_P3:=MAX(PWM_JOYY_L_UP,PWM_JOYX_R_UP);
			PWM_Y2_Target:=REAL_TO_UINT(UINT_TO_REAL(PWM_JOYY_L_UP)/1000*(PAR_Y1_PosFull-PAR_Y1_NegFull)+PAR_Y1_NegFull);
			PWM_Y1_Target:=REAL_TO_UINT(UINT_TO_REAL(PWM_JOYY_L_UP)/1000*(PAR_Y1_PosFull-PAR_Y1_NegFull)+PAR_Y1_NegFull);
			PWM_Y10_SET_Target:=REAL_TO_UINT(UINT_TO_REAL(PWM_JOYY_L_UP)/1000*(PAR_Valve1_PosFull-PAR_Valve1_NegFull)+PAR_Valve1_NegFull);
			PWM_Y8_SET_Target:=REAL_TO_UINT(UINT_TO_REAL(1000-PWM_JOYX_R_UP)/1000*(PAR_Valve1_PosFull-PAR_Valve1_NegFull)+PAR_Valve1_NegFull);
			PWM_Y7_SET_Target:=0;
			PWM_Y9_SET_Target:=0;
		END_IF	
	ELSIF PWM_JOYY_L_DOWN>10 THEN//主卷上提
		IF(PWM_JOYX_R_DOWN>10) THEN //动力头正转
			PWM_JOY_P2:=MAX(PWM_JOYY_L_DOWN,PWM_JOYX_R_DOWN);
			PWM_Y2_Target:=REAL_TO_UINT(UINT_TO_REAL(PWM_JOYY_L_DOWN)/1000*(PAR_Y1_PosFull-PAR_Y1_NegFull)+PAR_Y1_NegFull);
			PWM_Y1_Target:=REAL_TO_UINT(UINT_TO_REAL(PWM_JOYY_L_DOWN)/1000*(PAR_Y1_PosFull-PAR_Y1_NegFull)+PAR_Y1_NegFull);
			PWM_Y9_SET_Target:=REAL_TO_UINT(UINT_TO_REAL(PWM_JOYY_L_DOWN)/1000*(PAR_Valve1_PosFull-750)+750);
			PWM_Y7_SET_Target:=REAL_TO_UINT(UINT_TO_REAL(PWM_JOYY_L_DOWN)/1000*(PAR_Valve1_PosFull-750)+750);
			PWM_Y8_SET_Target:=0;
			PWM_Y10_SET_Target:=0;
		ELSIF PWM_JOYX_R_UP>10 THEN//动力头反转
			PWM_JOY_P1:=MAX(PWM_JOYY_L_DOWN,PWM_JOYX_R_UP);
			PWM_Y1_Target:=REAL_TO_UINT(UINT_TO_REAL(PWM_JOYY_L_DOWN)/1000*(PAR_Y1_PosFull-PAR_Y1_NegFull)+PAR_Y1_NegFull);
			PWM_Y2_Target:=REAL_TO_UINT(UINT_TO_REAL(PWM_JOYY_L_DOWN)/1000*(PAR_Y2_PosFull-PAR_Y2_NegFull)+PAR_Y2_NegFull);
			PWM_Y7_SET_Target:=REAL_TO_UINT(UINT_TO_REAL(PWM_JOYY_L_DOWN)/1000*(PAR_Valve1_PosFull-750)+750);
			PWM_Y9_SET_Target:=REAL_TO_UINT(UINT_TO_REAL(PWM_JOYY_L_DOWN)/1000*(PAR_Valve2_PosFull-750)+750);
			PWM_Y8_SET_Target:=0;
			PWM_Y10_SET_Target:=0;
		END_IF
	END_IF
ELSIF (MainWinch_move) AND (LeftMove_move OR RightMove_move) THEN
//主卷和行走复合动作 主泵1提供给主卷油
	IF PWM_JOYY_L_UP>10 THEN//主卷下放
		PWM_Y1_Target:=REAL_TO_UINT(UINT_TO_REAL(PWM_JOYY_L_UP)/1000*(PAR_Y1_PosFull-PAR_Y1_NegFull)+PAR_Y1_NegFull);
		PWM_Y10_SET_Target:=0;
		PWM_Y8_SET_Target:=PAR_Valve1_PosFull;
		PWM_Y7_SET_Target:=0;
		PWM_Y9_SET_Target:=0;
	ELSIF PWM_JOYY_L_DOWN>10 THEN//主卷上提
		PWM_Y1_Target:=REAL_TO_UINT(UINT_TO_REAL(PWM_JOYY_L_DOWN)/1000*(PAR_Y1_PosFull-PAR_Y1_NegFull)+PAR_Y1_NegFull);
		PWM_Y9_SET_Target:=0;
		PWM_Y7_SET_Target:=PAR_Valve1_PosFull;
		PWM_Y8_SET_Target:=0;
		PWM_Y10_SET_Target:=0;		
		PWM_Y19_SET:=0;
		IF(DI_LHandle_SB4)THEN
			PWM_Y20_SET:=600;
		ELSE
			PWM_Y20_SET:=0;
		END_IF
	END_IF
ELSE
		PWM_Y8_SET:=0;
		PWM_Y10_SET:=0;
		PWM_Y7_SET:=0;
		PWM_Y9_SET:=0;
		PWM_Y8_SET_Target:=0;
		PWM_Y10_SET_Target:=0;
		PWM_Y7_SET_Target:=0;
		PWM_Y9_SET_Target:=0;
END_IF
	
	
//主卷扬根据阀的开关调整斜坡值	
	IF(PWM_Y8_SET<1000  AND  PWM_Y8_SET>=900)THEN    //主卷下放斜坡值
			F_RAMP_mainwinch_down:=200;
	ELSIF(PWM_Y8_SET<900)THEN
			F_RAMP_mainwinch_down:=100;
	ELSE
			F_RAMP_mainwinch_down:=200;
	END_IF
		
	IF(PWM_Y7_SET<1000  AND  PWM_Y7_SET>=900)THEN  //主卷上提斜坡值
			F_RAMP_mainwinch_down:=300;
	ELSIF(PWM_Y7_SET<900  )THEN
			F_RAMP_mainwinch_down:=200;
	ELSE
			F_RAMP_mainwinch_down:=400;
	END_IF
		
RAMP7(
	IN:=WORD_TO_INT(PWM_Y7_SET_Target), 
	ASCEND:= R_RAMP_mainwinch, 
	DESCEND:= F_RAMP_mainwinch_up, 
	TIMEBASE:=TIMEBASE_mainwinch , 
	RESET:=FALSE , 
	OUT=>(PWM_Y7_SET_Target1));
IF(PWM_Y7_SET_Target1>=400) THEN
	Curve_input:=TO_UINT(PWM_Y7_SET_Target1 - 400);
	IF(Curve_input>900) THEN
		Curve_input:=900;
	END_IF
	curve7(input:=REAL_TO_UINT(UINT_TO_REAL(Curve_input)*72.8),Zero:=FALSE,Full:=FALSE,
		   PAR_Progression:=Curve_Par,OutputEnable:=TRUE);
	PWM_Y7_SET:=PAR_Valve1_NegFull + REAL_TO_UINT(UINT_TO_REAL(curve7.Output)/72.8);
ELSE
	PWM_Y7_SET:=0;
END_IF


RAMP8(
	IN:=WORD_TO_INT(PWM_Y8_SET_Target), 
	ASCEND:= R_RAMP_mainwinch, 
	DESCEND:= F_RAMP_mainwinch_down, 
	TIMEBASE:=TIMEBASE_mainwinch , 
	RESET:=FALSE , 
	OUT=>(PWM_Y8_SET_Target1));
IF(PWM_Y8_SET_Target1>=400) THEN
	Curve_input:=TO_UINT(PWM_Y8_SET_Target1 - 400);
	IF(Curve_input>900) THEN
		Curve_input:=900;
	END_IF
	curve8(input:=REAL_TO_UINT(UINT_TO_REAL(Curve_input)*72.8),Zero:=FALSE,Full:=FALSE,
		   PAR_Progression:=Curve_Par,OutputEnable:=TRUE);
	PWM_Y8_SET:=PAR_Valve1_NegFull + REAL_TO_UINT(UINT_TO_REAL(curve8.Output)/72.8);
ELSE
	PWM_Y8_SET:=0;
END_IF


RAMP9(
	IN:=WORD_TO_INT(PWM_Y9_SET_Target), 
	ASCEND:= R_RAMP_mainwinch, 
	DESCEND:= F_RAMP_mainwinch_up, 
	TIMEBASE:=TIMEBASE_mainwinch , 
	RESET:=FALSE , 
	OUT=>(PWM_Y9_SET_Target1));
IF(PWM_Y9_SET_Target1>=400) THEN
	Curve_input:=TO_UINT(PWM_Y9_SET_Target1 - 400);
	IF(Curve_input>900) THEN
		Curve_input:=900;
	END_IF
	curve9(input:=REAL_TO_UINT(UINT_TO_REAL(Curve_input)*72.8),Zero:=FALSE,Full:=FALSE,
		   PAR_Progression:=Curve_Par,OutputEnable:=TRUE);
	PWM_Y9_SET:=PAR_Valve1_NegFull + REAL_TO_UINT(UINT_TO_REAL(curve9.Output)/72.8);
ELSE
	PWM_Y9_SET:=0;
END_IF

RAMP10(
	IN:=WORD_TO_INT(PWM_Y10_SET_Target), 
	ASCEND:= R_RAMP_mainwinch, 
	DESCEND:= F_RAMP_mainwinch_down, 
	TIMEBASE:=TIMEBASE_mainwinch , 
	RESET:=FALSE , 
	OUT=>(PWM_Y10_SET_Target1));
IF(PWM_Y10_SET_Target1>=400) THEN
	Curve_input:=TO_UINT(PWM_Y10_SET_Target1 - 400);
	IF(Curve_input>900) THEN
		Curve_input:=900;
	END_IF
	curve10(input:=REAL_TO_UINT(UINT_TO_REAL(Curve_input)*72.8),Zero:=FALSE,Full:=FALSE,
		   PAR_Progression:=Curve_Par,OutputEnable:=TRUE);
	PWM_Y10_SET:=PAR_Valve1_NegFull + REAL_TO_UINT(UINT_TO_REAL(curve10.Output)/72.8);
ELSE
	PWM_Y10_SET:=0;
END_IF


IF(PWM_Y7_SET>1300)THEN
	PWM_Y7_SET :=1300;
END_IF
IF(PWM_Y8_SET>1300)THEN
	PWM_Y8_SET :=1300;
END_IF
IF(PWM_Y9_SET>1300)THEN
	PWM_Y9_SET :=1300;
END_IF
IF(PWM_Y10_SET>1300)THEN
	PWM_Y10_SET :=1300;
END_IF

IF(PWM_Y7_SET<=300)THEN
	PWM_Y7_SET :=0;
END_IF
IF(PWM_Y8_SET<=300)THEN
	PWM_Y8_SET :=0;
END_IF
IF(PWM_Y9_SET<=300)THEN
	PWM_Y9_SET :=0;
END_IF
IF(PWM_Y10_SET<=300)THEN
	PWM_Y10_SET :=0;
END_IF




(*主泵卸荷阀控制*)
		PWM_Y39_SET_Target:=MAX(PWM_Y8_SET_Target,PWM_Y7_SET_Target,PWM_Y12_SET_Tatget,PWM_Y11_SET_Tatget,PWM_Y3_SET,PWM_Y4_SET,PWM_Y15_SET_Target,PWM_Y16_SET_Target);
		PWM_Y40_SET_Target:=MAX(PWM_Y9_SET_Target,PWM_Y10_SET_Target,PWM_Y13_SET_Tatget,PWM_Y14_SET_Tatget,PWM_Y5_SET_Target,PWM_Y6_SET_Target,PWM_Y17_SET2,PWM_Y18_SET);
	(*卸荷动作缓冲*)
RAMP19(
	IN:=WORD_TO_INT(PWM_Y39_SET_Target), 
	ASCEND:= R_RAMP_xiehe, 
	DESCEND:= F_RAMP_xiehe, 
	TIMEBASE:=TIMEBASE_xiehe , 
	RESET:=FALSE , 
	OUT=>(PWM_Y39_SET_Target1));
IF(PWM_Y39_SET_Target1>=400) THEN
	Curve_input:=TO_UINT(PWM_Y39_SET_Target1 - 400);
	IF(Curve_input>900) THEN
		Curve_input:=900;
	END_IF
	curve19(input:=REAL_TO_UINT(UINT_TO_REAL(Curve_input)*72.8),Zero:=FALSE,Full:=FALSE,
		   PAR_Progression:=Curve_Par1,OutputEnable:=TRUE);
	PWM_Y39_SET:=PAR_Valve1_NegFull + REAL_TO_UINT(UINT_TO_REAL(curve19.Output)/72.8);
ELSE
	PWM_Y39_SET:=0;
END_IF


RAMP20(
	IN:=WORD_TO_INT(PWM_Y40_SET_Target), 
	ASCEND:= R_RAMP_xiehe, 
	DESCEND:= F_RAMP_xiehe, 
	TIMEBASE:=TIMEBASE_xiehe , 
	RESET:=FALSE , 
	OUT=>(PWM_Y40_SET_Target1));
IF(PWM_Y40_SET_Target1>=400) THEN
	Curve_input:=TO_UINT(PWM_Y40_SET_Target1 - 400);
	IF(Curve_input>900) THEN
		Curve_input:=900;
	END_IF
	curve20(input:=REAL_TO_UINT(UINT_TO_REAL(Curve_input)*72.8),Zero:=FALSE,Full:=FALSE,
		   PAR_Progression:=Curve_Par1,OutputEnable:=TRUE);
	PWM_Y40_SET:=PAR_Valve1_NegFull + REAL_TO_UINT(UINT_TO_REAL(curve20.Output)/72.8);
ELSE
	PWM_Y40_SET:=0;
END_IF

	//在行走时一个泵供油时,需要关闭另外一个 泵的起压阀
	IF PWM_Y37_SET>500 AND (NOT MainWinch_move) THEN
		PWM_Y39_SET:=0;
	END_IF
	
IF(PWM_Y39_SET>1300)THEN
	PWM_Y39_SET :=1300;
END_IF
IF(PWM_Y40_SET>1300)THEN
	PWM_Y40_SET :=1300;
END_IF

IF(PWM_Y39_SET<=300)THEN
	PWM_Y39_SET :=0;
END_IF
IF(PWM_Y40_SET<=300)THEN
	PWM_Y40_SET :=0;
END_IF

(*副卷扬动作*)
IF(ViceWinch_move)THEN
	IF PWM_JOYY_R_UP>10 THEN//副卷下放
		PWM_Y4_SET:=REAL_TO_UINT(UINT_TO_REAL(PWM_JOYY_R_UP)/1000*(1200-500)+500);
		PWM_Y3_SET:=0;
		IF(NOT MainWinch_move) OR (NOT PowerHead_move) THEN
			PWM_Y1_Target:=REAL_TO_UINT(UINT_TO_REAL(PWM_JOYY_R_UP)/1000*(PAR_KP-PAR_Y1_NegFull)+PAR_Y1_NegFull);
		END_IF
		
	ELSIF PWM_JOYY_R_DOWN>10 THEN//副卷上提
		PWM_Y3_SET:=REAL_TO_UINT(UINT_TO_REAL(PWM_JOYY_R_DOWN)/1000*(1200-500)+500);
		PWM_Y4_SET:=0;
		IF(NOT MainWinch_move) OR (NOT PowerHead_move) THEN
			PWM_Y1_Target:=REAL_TO_UINT(UINT_TO_REAL(PWM_JOYY_R_DOWN)/1000*(PAR_KP-PAR_Y1_NegFull)+PAR_Y1_NegFull);
		END_IF		
	END_IF
ELSE
	PWM_Y3_SET:=0;
	PWM_Y4_SET:=0;
END_IF

(*回转动作*)
//回转限制
IF  (CANO_DEPTH>980 AND  CANI_WorkModeSwitch) THEN
		Rotation_move:=FALSE;
END_IF
	
IF NOT DI_LHandle_SB7 THEN(*自动回转*) 
	IF  Rotation_move  OR DI_LHandle_SB2  THEN
		DOH_Y50_1 := TRUE;
		IF PWM_JOYX_L_UP>10 THEN// 右回转
			PWM_Y22_SET:=REAL_TO_UINT(UINT_TO_REAL(PWM_JOYX_L_UP)/1000*(PAR_ValveC_NegFull-PAR_Valve3_NegFull)+PAR_Valve3_NegFull);
			PWM_Y21_SET:=0;
		ELSIF PWM_JOYX_L_DOWN>10 THEN//左回转
			PWM_Y21_SET:=REAL_TO_UINT(UINT_TO_REAL(PWM_JOYX_L_DOWN)/1000*(PAR_ValveC_NegFull-PAR_Valve3_NegFull)+PAR_Valve3_NegFull);
			PWM_Y22_SET:=0;
		END_IF
	ELSE
		DOH_Y50_1:= FALSE;
		PWM_Y21_SET:=0;
		PWM_Y22_SET:=0;
	END_IF
ELSE
	DOH_Y50_1 := TRUE;
	IF(AUTO_ROTATION_VALVE>=0) THEN
		PWM_Y21_SET:=REAL_TO_UINT(INT_TO_REAL(ABS(AUTO_ROTATION_VALVE))*0.13);
	ELSE
		PWM_Y22_SET:=REAL_TO_UINT(INT_TO_REAL(ABS(AUTO_ROTATION_VALVE))*0.13);		
	END_IF
END_IF

//回转时警示灯响并且监控显示后界面
IF Rotation_move  OR DOH_Y50 THEN
	DOH_70:=TRUE;
	DOH_73:=TRUE;
	DOH_JK2:=TRUE;
ELSE
	DOH_70:=FALSE;
	DOH_73:=FALSE;
	DOH_JK2:=FALSE;
END_IF

//制动阀延时锁车
Rotation_late(IN:=DOH_Y50_1,PT:=T#2S);
IF  DOH_Y50_1 THEN
	DOH_Y50:=TRUE;
ELSE
	DOH_Y50:=Rotation_late.Q;
END_IF

(*加压动作*)
IF JiaYa_move THEN
	IF PWM_JOYY_R_UP>10 THEN//加压下
		PWM_Y23_SET_Taget:=REAL_TO_UINT(UINT_TO_REAL(PWM_JOYY_R_UP)/1000*(800-PAR_Valve3_NegFull)+PAR_Valve3_NegFull);
		PWM_Y24_SET_Taget:=0;
		
		IF(CANI_JiaYaFastSwitch OR DI_RHandle_SB7)THEN //加压快
			PWM_Y2_Target:=REAL_TO_UINT(UINT_TO_REAL(PWM_JOYY_R_UP)/1000*(500-300)+300);
			PWM_Y17_SET:=0;
			PWM_Y17_SET2:=0;
			PWM_Y18_SET_Taget:=1300;
		ELSE
			PWM_Y18_SET_Taget:=0;
		END_IF
		
	ELSIF PWM_JOYY_R_DOWN>10 THEN//加压上
		PWM_Y24_SET_Taget:=REAL_TO_UINT(UINT_TO_REAL(PWM_JOYY_R_DOWN)/1000*(800-PAR_Valve3_NegFull)+PAR_Valve3_NegFull);
		PWM_Y23_SET_Taget:=0;
		
		IF(CANI_JiaYaFastSwitch OR DI_RHandle_SB7)THEN //加压快
			PWM_Y2_Target:=REAL_TO_UINT(UINT_TO_REAL(PWM_JOYY_R_DOWN)/1000*(500-300)+300);
			PWM_Y17_SET:=800;
			PWM_Y17_SET2:=1300;
			PWM_Y18_SET:=0;
		ELSE
			PWM_Y18_SET:=0;
		END_IF
	END_IF
ELSE
	PWM_Y23_SET_Taget:=0;
	PWM_Y24_SET_Taget:=0;
	PWM_Y17_SET:=0;
	PWM_Y18_SET:=0;
	PWM_Y17_SET2:=0;
END_IF

RAMP22(
	IN:=WORD_TO_INT(PWM_Y23_SET_Taget), 
	ASCEND:= ASCEND_value, 
	DESCEND:= 5000, 
	TIMEBASE:=T#1000MS , 
	RESET:=FALSE , 
	OUT=>(PWM_Y23_SET_Taget1));
IF(PWM_Y23_SET_Taget1<310)THEN
		ASCEND_value:=6000;
ELSIF(PWM_Y23_SET_Taget1>=310 AND PWM_Y23_SET_Taget1<450)THEN
		ASCEND_value:=100;
ELSE
		ASCEND_value:=300;
END_IF
IF(PWM_Y23_SET_Taget1>=300) THEN
	Curve_input:=TO_UINT(PWM_Y23_SET_Taget1 - 300);
	IF(Curve_input>500) THEN
		Curve_input:=500;
	END_IF
	PWM_Y23_SET:=300 + Curve_input;
ELSE
	PWM_Y23_SET:=0;
END_IF

RAMP24(
	IN:=WORD_TO_INT(PWM_Y24_SET_Taget), 
	ASCEND:= 500, 
	DESCEND:= 500, //500-6000
	TIMEBASE:=T#300MS , 
	RESET:=FALSE , 
	OUT=>((PWM_Y24_SET)));
(*IF(PWM_Y24_SET_Taget1>=300) THEN
	Curve_input:=TO_UINT(PWM_Y24_SET_Taget1 - 300);
	IF(Curve_input>500) THEN
		Curve_input:=500;
	END_IF
	PWM_Y24_SET:=300 + Curve_input;
ELSE
	PWM_Y24_SET:=0;
END_IF*)



RAMP23(
	IN:=WORD_TO_INT(PWM_Y18_SET_Taget), 
	ASCEND:= ASCEND_value2, 
	DESCEND:= 5000, 
	TIMEBASE:=T#1000MS , 
	RESET:=FALSE , 
	OUT=>(PWM_Y18_SET_Taget1));
IF(PWM_Y18_SET_Taget1<610)THEN
		ASCEND_value2:=6000;
ELSE
	ASCEND_value2:=150;
END_IF	

IF(PWM_Y18_SET_Taget1>=600) THEN
	Curve_input:=TO_UINT(PWM_Y18_SET_Taget1 - 600);
	IF(Curve_input>700) THEN
		Curve_input:=700;
	END_IF
	PWM_Y18_SET:=600 + Curve_input;
ELSE
	PWM_Y18_SET:=0;
END_IF

(*PWM_Y23_SET:=PWM_Y23_SET_Taget;*)
IF JiaYa_move THEN
	IF PWM_JOYY_R_DOWN>10 THEN
		PWM_Y23_SET_Taget:=0;
		PWM_Y23_SET_Taget1:=0;
		PWM_Y23_SET:=0;
		PWM_Y18_SET_Taget1:=0;
		PWM_Y18_SET_Taget:=0;
		PWM_Y18_SET:=0;
	END_IF
END_IF

//加压限压
IF(CANI_DongLiTouPressLimitSwitch)THEN
	PWM_Y63_SET:=PAR_ValveD_PosFull;
ELSE
	PWM_Y63_SET:=0;
END_IF
		
(*平举动作*)
IF  BianFu_move THEN
	IF PWM_JOYY_R_UP>10 THEN//变幅下
		PWM_Y25_SET:=REAL_TO_UINT(UINT_TO_REAL(PWM_JOYY_R_UP)/1000*(PAR_Valve3_PosFull-PAR_Valve3_NegFull)+PAR_Valve3_NegFull);
		PWM_Y26_SET:=0;
	ELSIF PWM_JOYY_R_DOWN>10 THEN//变幅上
		PWM_Y26_SET:=REAL_TO_UINT(UINT_TO_REAL(PWM_JOYY_R_DOWN)/1000*(PAR_Valve3_PosFull-PAR_Valve3_NegFull)+PAR_Valve3_NegFull);
		PWM_Y25_SET:=0;
	END_IF
ELSE
	PWM_Y25_SET:=0;
	PWM_Y26_SET:=0;
END_IF

(*张紧等切换油缸动作*)
IF  LvZhang_move THEN
	IF(NOT CANI_LvDaiShenSuoSwitch)THEN
		IF PWM_JOYX_R_UP>10 THEN
			PWM_Y31_SET:=REAL_TO_UINT(UINT_TO_REAL(PWM_JOYX_R_UP)/1000*(PAR_Valve3_PosFull-PAR_Valve3_NegFull)+PAR_Valve3_NegFull);
			PWM_Y32_SET:=0;
			PWM_Y19_SET:=0;
			PWM_Y20_SET:=0;
		ELSIF PWM_JOYX_R_DOWN>10 THEN
			PWM_Y32_SET:=REAL_TO_UINT(UINT_TO_REAL(PWM_JOYX_R_DOWN)/1000*(PAR_Valve3_PosFull-PAR_Valve3_NegFull)+PAR_Valve3_NegFull);
			PWM_Y31_SET:=0;
			PWM_Y19_SET:=0;
			PWM_Y20_SET:=0;
		ELSE
			PWM_Y31_SET:=0;
			PWM_Y32_SET:=0;
			PWM_Y19_SET:=0;
			PWM_Y20_SET:=0;
		END_IF
	ELSE
		IF PWM_JOYX_R_UP>10 THEN
			PWM_Y19_SET:=REAL_TO_UINT(UINT_TO_REAL(PWM_JOYX_R_UP)/1000*(PAR_Valve3_PosFull-PAR_Valve3_NegFull)+PAR_Valve3_NegFull);
			PWM_Y20_SET:=0;
			PWM_Y31_SET:=0;
			PWM_Y32_SET:=0;
		ELSIF PWM_JOYX_R_DOWN>10 THEN
			PWM_Y20_SET:=REAL_TO_UINT(UINT_TO_REAL(PWM_JOYX_R_DOWN)/1000*(PAR_Valve3_PosFull-PAR_Valve3_NegFull)+PAR_Valve3_NegFull);
			PWM_Y19_SET:=0;
			PWM_Y31_SET:=0;
			PWM_Y32_SET:=0;
		ELSE
			PWM_Y31_SET:=0;
			PWM_Y32_SET:=0;
			PWM_Y19_SET:=0;
			PWM_Y20_SET:=0;
		END_IF
	END_IF
ELSE
	PWM_Y31_SET:=0;
	PWM_Y32_SET:=0;
	PWM_Y19_SET:=0;
	PWM_Y20_SET:=0;
END_IF


IF(CANI_ETouYouGangSwitch) THEN//支腿/鹅头油缸切换
	DOH_Y52:=TRUE;
ELSE
	DOH_Y52:=FALSE;
END_IF

//主卷动作及浮动时开锁
IF  MainWinch_move OR DOH_Y55 THEN
	DOH_Y53 := TRUE;
	DOH_Y64:=TRUE;
	GVL_SaveEngine.Y74:=TRUE;
ELSE
	DOH_Y53 := FALSE;	
	DOH_Y64:=FALSE;
	GVL_SaveEngine.Y74:=FALSE;
END_IF

(*主泵功率控制20230706*)
//区分发动机转速
MainPump_Pressure_Taget1450:=PAR_NegFull_x;
MainPump_Pressure_Taget1600:=PAR_PosFull_x;
MainPump_Pressure_Taget1750:=PAR_Zero_x;

IF EngineSpeedTarget<=1080 THEN SPEED_CASE:=1;
ELSIF EngineSpeedTarget>1080 AND EngineSpeedTarget<=1300 THEN SPEED_CASE:=2;
ELSIF EngineSpeedTarget>1300 AND EngineSpeedTarget<=1520 THEN SPEED_CASE:=3;
ELSIF EngineSpeedTarget>1520 AND EngineSpeedTarget<=1680 THEN SPEED_CASE:=4;
ELSIF EngineSpeedTarget>1680 AND EngineSpeedTarget<=1820 THEN SPEED_CASE:=5;
ELSIF EngineSpeedTarget>1820 THEN SPEED_CASE:=6;;END_IF
//不同转速下的发动机最大功率
CASE SPEED_CASE OF
1:  Enginer_Power:=135;
2:  Enginer_Power:=174;
3:  Enginer_Power:=200;
4:  Enginer_Power:=230;
5:  Enginer_Power:=250;
6:  Enginer_Power:=261;
END_CASE
//不同转速下的压力值
IF(CANO_Fubeng_Press>100)THEN
	CASE SPEED_CASE OF
		1:MainPump_Pressure_Taget:=MainPump_Pressure_Taget1000-HELIU_Press_Target1000;
		2:MainPump_Pressure_Taget:=MainPump_Pressure_Taget1200-HELIU_Press_Target1200;
		3:MainPump_Pressure_Taget:=MainPump_Pressure_Taget1450-HELIU_Press_Target1400;
		4:MainPump_Pressure_Taget:=MainPump_Pressure_Taget1600-HELIU_Press_Target1600;
		5:MainPump_Pressure_Taget:=MainPump_Pressure_Taget1750-HELIU_Press_Target1800;
		6:MainPump_Pressure_Taget:=MainPump_Pressure_Taget1900-HELIU_Press_Target1900;
	END_CASE
ELSE
	CASE SPEED_CASE OF
		1:MainPump_Pressure_Taget:=MainPump_Pressure_Taget1000;
		2:MainPump_Pressure_Taget:=MainPump_Pressure_Taget1200;
		3:MainPump_Pressure_Taget:=MainPump_Pressure_Taget1450;
		4:MainPump_Pressure_Taget:=MainPump_Pressure_Taget1600;
		5:MainPump_Pressure_Taget:=MainPump_Pressure_Taget1750;
		6:MainPump_Pressure_Taget:=MainPump_Pressure_Taget1900;
	END_CASE		
END_IF
IF( CANI_ECOSwitch) THEN
	CASE SPEED_CASE OF
		1:MainPump_Pressure_Taget:=MainPump_Pressure_Taget1000-ECO_Press_Target1000;
		2:MainPump_Pressure_Taget:=MainPump_Pressure_Taget1200-ECO_Press_Target1200;
		3:MainPump_Pressure_Taget:=MainPump_Pressure_Taget1450-ECO_Press_Target1400;
		4:MainPump_Pressure_Taget:=MainPump_Pressure_Taget1600-ECO_Press_Target1600;
		5:MainPump_Pressure_Taget:=MainPump_Pressure_Taget1750-ECO_Press_Target1800;
		6:MainPump_Pressure_Taget:=MainPump_Pressure_Taget1900-ECO_Press_Target1900;
	END_CASE
END_IF
MainPump_Pressure:=CANO_MainPUMP_Press1+CANO_MainPUMP_Press2;
//消除滤波
MainPump_Pressure_Subtract:= UINT_TO_INT(MainPump_Pressure-MainPump_Pressure_last1);

TIME_200ms(IN:=NOT TIME_200ms.Q,PT:=T#400MS);

IF(TIME_200ms.Q)THEN
	CANI_JOYX_R_last:=CANI_JOYX_R;
END_IF
Sub_Joyx_r:=UINT_TO_INT(CANI_JOYX_R_last) - UINT_TO_INT(CANI_JOYX_R);
IF(Sub_Joyx_r<-1200 OR Sub_Joyx_r>1200) THEN
	Joyx_change_bool:=TRUE;
	
END_IF

IF(CANI_JOYX_R=2500)THEN
	tempbool:=TRUE;
ELSE
	tempbool:=FALSE;
END_IF

TIME_1000_1ms(in:=tempbool,PT:=T#500MS);
IF(TIME_1000_1ms.Q)THEN
	JOY_PAOTU:=FALSE;
END_IF

TIME_400ms(IN:=Joyx_change_bool,PT:=T#10MS);
IF(TIME_400ms.Q) THEN
	Joyx_change_bool:=FALSE;
END_IF



//大范围波动
IF MainPump_Pressure_Subtract>270 OR MainPump_Pressure_Subtract<-270 THEN
	Subtract:=TRUE;
ELSE
	Subtract:=FALSE;	
END_IF
	TIME_LvBo4(IN:=Subtract,PT:=T#10MS);
	
IF(TIME_LvBo4.Q) AND (CANO_MainPUMP_Press1>210) THEN 
		MainPump_Pressure_ChangeBool1:=TRUE;
END_IF
	TIME_LvBo1(IN:=MainPump_Pressure_ChangeBool1,PT:=T#2S);
IF(TIME_LvBo1.Q) THEN
	MainPump_Pressure_ChangeBool1 :=FALSE;
END_IF

IF(MainPump_Pressure_ChangeBool1) AND (MainPump_Pressure>MainPump_Pressure_last1) THEN 
	MainPump_Pressure_last1:=MainPump_Pressure;
END_IF

//小范围波动
t_powertime:=TO_TIME(PAR_DeadBand_x);
IF (NOT MainPump_Pressure_ChangeBool1) THEN
	IF(MainPump_Pressure_Subtract>40 OR MainPump_Pressure_Subtract<-40)THEN 
		MainPump_Pressure_ChangeBool:=TRUE;
	ELSE
		MainPump_Pressure_ChangeBool:=FALSE;
	END_IF

	TIME_LvBo2(IN:=MainPump_Pressure_ChangeBool,PT:=t_powertime);
	IF(TIME_LvBo2.Q )THEN
		MainPump_Pressure_last1:=MainPump_Pressure;
	END_IF	
END_IF


IF PowerHead_move AND NOT(MainWinch_move) THEN
		JianGE2:=0.005;
ELSE
	IF(EngineSpeedTarget>1000 AND EngineSpeedTarget<1300)THEN
		JianGE2:=0.005;
	ELSE
		JianGE2:=0.005;
	END_IF
END_IF
	
IF MainPump_Pressure_last1>MainPump_Pressure_Taget THEN
	Pressure_Coe_Taget:=UINT_TO_REAL(MainPump_Pressure_Taget)/UINT_TO_REAL(MainPump_Pressure_last1);(*压力系数*)
ELSE
	Pressure_Coe_Taget:=1;
END_IF
Pressure_Coe := Pressure_Coe_Taget;


IF MainPump_Pressure_last1>MainPump_Pressure_Taget  THEN
	IF(PWM_Y1_Target>=PAR_Y1_1_NegFull)THEN
		PWM_Y1_Target_OutPut:=REAL_TO_UINT(UINT_TO_REAL(PWM_Y1_Target-PAR_Y1_1_NegFull)*Pressure_Coe+PAR_Y1_1_NegFull);
	END_IF
	IF(PWM_Y2_Target>=PAR_Y1_1_NegFull)THEN
		PWM_Y2_Target_OutPut:=REAL_TO_UINT(UINT_TO_REAL(PWM_Y2_Target-PAR_Y1_1_NegFull)*Pressure_Coe+PAR_Y1_1_NegFull);
	END_IF
ELSE
	PWM_Y1_Target_OutPut:=PWM_Y1_Target;
	PWM_Y2_Target_OutPut:=PWM_Y2_Target;
END_IF

IF(EngineSpeedTarget>CANO_SPEED AND CANO_SPEED>400)THEN
	EngineSpeedSub:=EngineSpeedTarget - CANO_SPEED;
ELSE
	EngineSpeedSub:=0;
END_IF

IF(PWM_Y1_Target_OutPut<300)THEN PWM_Y1_Target_OutPut:=300;END_IF	
IF(PWM_Y2_Target_OutPut<300)THEN PWM_Y2_Target_OutPut:=300;END_IF

RAMP15_IN:=PWM_Y1_Target_OutPut;
RAMP16_IN:=PWM_Y2_Target_OutPut;


IF MainWinch_move  OR  LeftMove_move OR RightMove_move THEN  
	TIMEBASE_pump:=T#1000MS;
	TIMEBASE_xiehe:=T#500MS;
ELSE
	TIMEBASE_pump:=T#600MS;
	TIMEBASE_xiehe:=T#300MS;
END_IF
t_PowerHead_move(IN:= MainWinch_move,PT:=T#4S);
IF t_PowerHead_move.Q THEN
	F_RAMP_pump:=x_t_PowerHead_move;
	R_RAMP_pump:=x2_t_PowerHead_move;
ELSE
       CASE SPEED_CASE OF
                1:F_RAMP_pump:=1500; R_RAMP_pump:=100;                  
                2: 		IF MainWinch_move AND (JiaYa_move OR CANO_JiayaPressure>80)  THEN    //3泵同时起压时，降低主泵的加载速度，避免掉速熄火
                                F_RAMP_pump:=1500; R_RAMP_pump:=100;
                        ELSE
                                F_RAMP_pump:=1500; R_RAMP_pump:=100;//从200降
                                IF  PWM_JOYY_L_UP>10 THEN
                                 F_RAMP_pump:=1500; R_RAMP_pump:=200;
                                END_IF
                        END_IF            
                3:
                        IF MainWinch_move AND (JiaYa_move OR CANO_JiayaPressure>80)  THEN    //3泵同时起压时，降低主泵的加载速度，避免掉速熄火
                                F_RAMP_pump:=1500; R_RAMP_pump:=150;
                        ELSE
                                F_RAMP_pump:=1500; R_RAMP_pump:=TO_INT(PAR_NegFull_y);
                                IF  PWM_JOYY_L_UP>10 THEN
                                 F_RAMP_pump:=1500; R_RAMP_pump:=300;
                                END_IF
                        END_IF                
                4:
                        IF MainWinch_move AND (JiaYa_move OR CANO_JiayaPressure>80)  THEN
                                F_RAMP_pump:=1500; R_RAMP_pump:=150;
                        ELSE
                                F_RAMP_pump:=1500; R_RAMP_pump:=TO_INT(PAR_PosFull_y);//从200降
                                IF  PWM_JOYY_L_UP>10 THEN
                                 F_RAMP_pump:=1500; R_RAMP_pump:=300;
                                END_IF
                        END_IF                                
                5:
                        IF MainWinch_move AND (JiaYa_move OR CANO_JiayaPressure>80)  THEN
                                F_RAMP_pump:=1500; R_RAMP_pump:=200;
                        ELSE
                                F_RAMP_pump:=1500; R_RAMP_pump:=TO_INT(PAR_Zero_y);
                                IF  PWM_JOYY_L_UP>10 THEN
                                 F_RAMP_pump:=1500; R_RAMP_pump:=300;
                                END_IF
                        END_IF                        
                6:		IF MainWinch_move AND (JiaYa_move OR CANO_JiayaPressure>80)  THEN
                                F_RAMP_pump:=1500; R_RAMP_pump:=200;
                        ELSE
                                F_RAMP_pump:=1500; R_RAMP_pump:=200;
                                IF  PWM_JOYY_L_UP>10 THEN
                                 F_RAMP_pump:=1500; R_RAMP_pump:=300;
                                END_IF
                        END_IF               
         END_CASE	
END_IF

RAMP15(
	IN:=UINT_TO_INT(RAMP15_IN), 
	ASCEND:= R_RAMP_pump, 
	DESCEND:= F_RAMP_pump, 
	TIMEBASE:=TIMEBASE_pump , 
	RESET:=FALSE , 
	OUT=>(PWM_Y1_SET));
	
RAMP16(
	IN:=UINT_TO_INT(RAMP16_IN), 
	ASCEND:= R_RAMP_pump, 
	DESCEND:= F_RAMP_pump, 
	TIMEBASE:=TIMEBASE_pump , 
	RESET:=FALSE , 
	OUT=>(PWM_Y2_SET));

IF (NOT Rotation_move) AND (NOT MainWinch_move) AND (NOT PowerHead_move)
		AND (NOT JiaYa_move) AND (NOT ViceWinch_move)
		AND (NOT LeftMove_move) AND (NOT RightMove_move)  THEN
	PWM_Y1_Target:=0;
	PWM_Y2_Target:=0;
END_IF


IF PWM_Y1_SET<TO_INT(PAR_Y1_1_NegFull )THEN
	PWM_Y1_SET:=TO_INT(PAR_Y1_1_NegFull);
END_IF

IF PWM_Y2_SET<TO_INT(PAR_Y1_1_NegFull )THEN
	PWM_Y2_SET:=TO_INT(PAR_Y1_1_NegFull);
END_IF

IF(PWM_Y1_SET>1000) THEN
	PWM_Y1_SET := 300;
END_IF

IF(PWM_Y2_SET>1000) THEN
	PWM_Y2_SET := 300;
END_IF
(*电控马达动力头变量控制*)
(*
DonglitouPressureSub:=UINT_TO_INT(CANO_DonglitouPressure - CANO_DonglitouPressure_last);
//只需小范围波动滤波
	IF(DonglitouPressureSub>10 OR DonglitouPressureSub<-10)THEN 
		DonglitouPressure_ChangeBool:=TRUE;
	ELSE
		DonglitouPressure_ChangeBool:=FALSE;
	END_IF

	TIME_LvBo3(IN:=DonglitouPressure_ChangeBool,PT:=T#500MS);
	IF(TIME_LvBo3.Q )THEN
		CANO_DonglitouPressure_last:=CANO_DonglitouPressure;
	END_IF	
IF(PWM_JOYX_R_UP>10 OR PWM_JOYX_R_DOWN>10)THEN
	IF(CANO_DonglitouPressure_last>260) THEN
	PWM_Y34_SET_Target :=380;   
	ELSIF(CANO_DonglitouPressure_last>240) THEN   
	PWM_Y34_SET_Target :=508;  
	ELSIF(CANO_DonglitouPressure_last>220) THEN   
	PWM_Y34_SET_Target :=605;  
	ELSIF(CANO_DonglitouPressure_last>200) THEN   
	PWM_Y34_SET_Target :=703;  
	ELSIF(CANO_DonglitouPressure_last>180) THEN   
	PWM_Y34_SET_Target :=801;  
	ELSIF(CANO_DonglitouPressure_last>160) THEN   
	PWM_Y34_SET_Target :=899;  
	ELSE
	PWM_Y34_SET_Target :=1100;  
	END_IF
ELSE
	PWM_Y34_SET_Target :=1100;  
END_IF

IF(CANO_DonglitouPressure<20) THEN
	JianGE22:=10;
ELSE
	JianGE22:=1.5;
END_IF
IF PWM_Y34_SET>PWM_Y34_SET_Target THEN
	PWM_Y34_SET := REAL_TO_UINT(UINT_TO_REAL(PWM_Y34_SET)-JianGE22);
END_IF

IF(PWM_Y34_SET<=PWM_Y34_SET_Target) THEN
	PWM_Y34_SET:=REAL_TO_UINT(UINT_TO_REAL(PWM_Y34_SET)+JianGE22);
END_IF


//H.M.L档
IF(CANI_DonglitouMSwitch) THEN
	IF(CANO_DonglitouPressure>280) THEN
		PWM_Y34_SET_Target :=380;  
	ELSIF(CANO_DonglitouPressure>270) THEN   
		PWM_Y34_SET_Target :=459;  
	ELSIF(CANO_DonglitouPressure>260) THEN   
		PWM_Y34_SET_Target :=508;  
	ELSIF(CANO_DonglitouPressure>250) THEN   
		PWM_Y34_SET_Target :=557;  
	ELSIF(CANO_DonglitouPressure>240) THEN   
		PWM_Y34_SET_Target :=605;  
	ELSIF(CANO_DonglitouPressure>230) THEN   
		PWM_Y34_SET_Target :=654;  
	ELSE
		PWM_Y34_SET_Target:=703;
	END_IF
END_IF

IF(CANI_DonglitouHSwitch) THEN
	PWM_Y34_SET_Target := 200;
END_IF

IF(DIH_SA15)THEN
	IF(PWM_Y34_SET_Target<600)THEN
		PWM_Y34_SET_Target:=600;
	END_IF
END_IF

IF PWM_Y34_SET>=PWM_Y34_SET_Target THEN
	PWM_Y34_SET := PWM_Y34_SET_Target;
END_IF

IF DIL_SQ3 THEN
	PWM_Y34_SET:=200;
END_IF

IF(PWM_Y34_SET>2000) THEN
	PWM_Y34_SET := 2000;
END_IF
*)
//液控马达
//动力头调速
Rtrig_d1(CLK:=CANI_DonglitouADDSwitch);
Rtrig_d2(CLK:=CANI_DonglitouSUBSwitch);
IF (Rtrig_d1.Q AND DI_LHandle_SB1 )THEN
	IF(CANI_DonglitouHSwitch AND NOT CANI_DonglitouLSwitch AND NOT CANI_DonglitouMSwitch)THEN
		PAR_MotorChioce_H_PWM:=PAR_MotorChioce_H_PWM+10;
	ELSIF(CANI_DonglitouMSwitch AND NOT CANI_DonglitouLSwitch AND NOT CANI_DonglitouHSwitch)THEN
		PAR_MotorChioce_M_PWM:=PAR_MotorChioce_M_PWM+10;
	ELSE
		PAR_MotorChioce_L_PWM:=PAR_MotorChioce_L_PWM+10;
	END_IF
ELSIF(Rtrig_d2.Q AND DI_LHandle_SB1)THEN
	IF(CANI_DonglitouHSwitch AND NOT CANI_DonglitouLSwitch AND NOT CANI_DonglitouMSwitch)THEN
		IF PAR_MotorChioce_H_PWM<20 THEN
			PAR_MotorChioce_H_PWM:=20;
		END_IF
		PAR_MotorChioce_H_PWM:=PAR_MotorChioce_H_PWM-10;
	ELSIF(CANI_DonglitouMSwitch AND NOT CANI_DonglitouLSwitch AND NOT CANI_DonglitouHSwitch)THEN
		IF PAR_MotorChioce_M_PWM<20 THEN
			PAR_MotorChioce_M_PWM:=20;
		END_IF
		PAR_MotorChioce_M_PWM:=PAR_MotorChioce_M_PWM-10;
	ELSE

		IF PAR_MotorChioce_L_PWM<20 THEN
			PAR_MotorChioce_L_PWM:=20;
		END_IF
		PAR_MotorChioce_L_PWM:=PAR_MotorChioce_L_PWM-10;
	END_IF
END_IF

	IF(CANI_DonglitouHSwitch AND NOT CANI_DonglitouLSwitch AND NOT CANI_DonglitouMSwitch)THEN
		PWM_Y34_SET:=PAR_MotorChioce_H_PWM;
	ELSIF(CANI_DonglitouMSwitch AND NOT CANI_DonglitouLSwitch AND NOT CANI_DonglitouHSwitch)THEN
		PWM_Y34_SET:=PAR_MotorChioce_M_PWM;
	ELSE
		PWM_Y34_SET:=PAR_MotorChioce_L_PWM;
	END_IF

PressLvBo_TON(IN:=CANO_ZhuJuanPressure>310,PT:=T#300MS);
PressLvBo_TON1(IN:=CANO_ZhuJuanPressure>290 AND CANO_ZhuJuanPressure<=310,PT:=T#300MS);
PressLvBo_TON2(IN:=CANO_ZhuJuanPressure>270 AND CANO_ZhuJuanPressure<=290,PT:=T#300MS);
PressLvBo_TON3(IN:=CANO_ZhuJuanPressure>250 AND CANO_ZhuJuanPressure<=270,PT:=T#300MS);
IF(CANO_ZhuJuanPressure>310 AND PressLvBo_TON.Q) OR P31_Flag THEN
        PWM_Y33_SET_Target :=230;   //排量200
        P31_Flag:=TRUE;
        IF (CANO_ZhuJuanPressure<270) THEN
                P31_Flag:=FALSE;        
        END_IF
ELSIF(CANO_ZhuJuanPressure>290 AND PressLvBo_TON1.Q) OR P29_Flag THEN   
        PWM_Y33_SET_Target :=267;   //排量180
        P29_Flag:=TRUE; 
        IF (CANO_ZhuJuanPressure<250) THEN
                P29_Flag:=FALSE; 
        END_IF
ELSIF(CANO_ZhuJuanPressure>270 AND PressLvBo_TON2.Q) OR P27_Flag THEN   
        PWM_Y33_SET_Target :=304;  //排量160
        P27_Flag:=TRUE;
        IF (CANO_ZhuJuanPressure<230) THEN
                P27_Flag:=FALSE; 
        END_IF
ELSIF(CANO_ZhuJuanPressure>250 AND PressLvBo_TON3.Q) OR P25_Flag THEN //压力小于270   
        PWM_Y33_SET_Target :=340;  //排量140
        P25_Flag:=TRUE; 
        IF (CANO_ZhuJuanPressure<210) THEN
                P25_Flag:=FALSE; 
        END_IF
ELSE //(CANO_ZhuJuanPressure<=250) THEN
        PWM_Y33_SET_Target :=370;
END_IF

IF NOT MainWinch_move THEN
    P25_Flag:=FALSE;
    P27_Flag:=FALSE;
    P29_Flag:=FALSE; 
    P31_Flag:=FALSE;        
END_IF     

  
//PWM_Y33_SET_Target:=Y33_1;

IF BiaoZHI_MainWinchUp THEN  //单主卷下放370马达电流
 	PWM_Y33_SET_Target:=370;
END_IF


IF PWM_Y33_SET>=PWM_Y33_SET_Target THEN
	PWM_Y33_SET := PWM_Y33_SET_Target;
END_IF
	
IF(PWM_Y33_SET<PWM_Y33_SET_Target) THEN
	PWM_Y33_SET:=REAL_TO_UINT(UINT_TO_REAL(PWM_Y33_SET)+JianGE6);
END_IF

IF DIL_SQ3 THEN
	PWM_Y33_SET:=0;
END_IF
//动力头抛土
(******************抛土控制******************)
(*自动抛土*)
	IF DI_RHandle_SB6 AND PowerHead_move THEN
		IF CANO_JiayaPressure>80 OR Rotation_move THEN     //抛土模式做了延时，防止3泵工作熄火
			PWM_Y1_SET:=450;//此值要确认抛土效果 
			PWM_Y2_SET:=450;
		ELSE
			PWM_Y1_SET:=UINT_TO_INT(PAR_ValveC_PosFull);
			PWM_Y2_SET:=UINT_TO_INT(PAR_ValveC_PosFull);
		END_IF
		PWM_Y39_SET:=1300;
		PWM_Y40_SET:=1300;
		DonglitouBlink(ENABLE:=TRUE,TIMELOW:=T#300MS,TIMEHIGH:=T#300MS);
		IF DonglitouBlink.OUT THEN
			PWM_Y12_SET:=PAR_Valve1_PosFull;
			PWM_Y14_SET:=PAR_Valve2_PosFull;
			PWM_Y61_SET:=PAR_Valve1_PosFull;
			PWM_Y11_SET:=0;
			PWM_Y13_SET:=0;
			PWM_Y60_SET:=0;
		ELSE
			DonglitouBlink_biaozhi:=FALSE;
			PWM_Y12_SET:=0;
			PWM_Y14_SET:=0;
			PWM_Y61_SET:=0;
			PWM_Y11_SET:=PAR_Valve1_PosFull;
			PWM_Y13_SET:=PAR_Valve2_PosFull;
			PWM_Y60_SET:=PAR_Valve1_PosFull;
		END_IF
	END_IF
	
	
	(*主卷自动抖土*)
	(*IF DI_LHandle_SB2 AND PowerHead_move THEN
		PWM_Y1_SET:=TO_INT(PAR_ValveD_PosFull);
		PWM_Y2_SET:=TO_INT(PAR_ValveD_PosFull);
		PWM_Y39_SET:=1200;
		PWM_Y40_SET:=1200;
		DonglitouBlink(ENABLE:=TRUE,TIMELOW:=T#400MS,TIMEHIGH:=T#400MS);
		IF DonglitouBlink.OUT THEN
			PWM_Y7_SET:=PAR_Valve1_PosFull;
			PWM_Y9_SET:=PAR_Valve2_PosFull;
		ELSE
			PWM_Y7_SET:=0;
			PWM_Y9_SET:=0;
		END_IF
	END_IF*)



(*冷却风扇控制*)
IF NOT CANI_ColdFunSwitch  THEN
	IF(CANO_Hyd_Tem>60)THEN
		PWM_Y49_SET := PAR_ValveD_NegFull;
	END_IF
	
	IF(CANO_Hyd_Tem<60)THEN
		PWM_Y49_SET := 0;		
	END_IF
ELSE
	PWM_Y49_SET := PAR_ValveD_NegFull;
END_IF

(*主卷浮动*)
IF((DIH_SA8 OR DI_LHandle_SB3 OR CANI_Button_FloatSwitch) AND CANI_MaiWinFloatSwitch AND (NOT DIL_SQ3)) THEN
	DOH_Y55:=TRUE;
	DOH_Y56:=TRUE;
ELSE
	DOH_Y55:=FALSE;
	DOH_Y56:=FALSE;
END_IF

(*主卷开锁*)
(*IF MainWinch_move AND (NOT PowerHead_move )AND (PWM_JOYY_L_UP<500 AND PWM_JOYY_L_DOWN=0) AND CANO_ZhuJuanPressure<100 THEN
	DOH_Y56:=TRUE;
END_IF*)

IF(UIGroupVoltage0<2000 OR UIGroupVoltage1<2000 OR UIGroupVoltage2<2000 
   OR UIGroupVoltage3<2000 OR UIGroupVoltage4<2000 OR UIGroupVoltage5<2000) THEN
	reset111:=TRUE;
ELSE
	reset111:=FALSE;
END_IF
(*
IF Paotu_Modle THEN
	PWM_Y1_SET:=UINT_TO_INT(testpaotu);//PAR_ValveC_PosFull
	PWM_Y2_SET:=UINT_TO_INT(testpaotu);
END_IF
*)

IF Paotu_Modle THEN
	IF CANO_JiayaPressure>80 OR Rotation_move THEN     //抛土模式做了延时，防止3泵工作熄火
		PWM_Y1_SET:=450;//此值要确认抛土效果 
		PWM_Y2_SET:=450;
	ELSE
		PWM_Y1_SET:=UINT_TO_INT(PAR_ValveC_PosFull);
		PWM_Y2_SET:=UINT_TO_INT(PAR_ValveC_PosFull);
	END_IF
	PWM_Y39_SET:=1300;
	PWM_Y40_SET:=1300;
END_IF

END_PROGRAM

// StandardPLC/Application/MOVE/curve_quxian
FUNCTION_BLOCK curve_quxian
VAR_INPUT
	input:UINT;
	Zero:BOOL;
	Full:BOOL;
	PAR_Progression:SINT;
	OutputEnable:BOOL;
END_VAR

VAR_OUTPUT
	Output:UINT;
END_VAR
VAR
	x:REAL;
	y:REAL;
	y1:REAL;
	y2:REAL;
	y3:REAL;
END_VAR

IF(OutputEnable)THEN
	
	x:=UINT_TO_REAL(input)/65535;
	
	IF(PAR_Progression>=0)THEN
		y1:=((x*x*x*SINT_TO_REAL(PAR_Progression)/100.0+(x*(100.0-SINT_TO_REAL(PAR_Progression)))/100.0));
		Output:=REAL_TO_UINT(y1*65535.0);
	ELSIF(PAR_Progression<0)THEN
		y2:=(1-((1-x)*(1-x)*(1-x)*(-SINT_TO_REAL(PAR_Progression))/100.0+(1-x)*(100+SINT_TO_REAL(PAR_Progression))/100.0));
		Output:=REAL_TO_UINT(y2*65535.0);
	END_IF
END_IF
IF(zero)THEN
	Output:=0;
END_IF
IF(Full) AND (NOT zero) THEN
	Output:=65535;
END_IF

IF(input>65535) THEN
	input:=65535;
END_IF

END_FUNCTION_BLOCK

// StandardPLC/Application/SaveEngine/SaveEngine
PROGRAM SaveEngine
VAR
END_VAR

MainWinTension_Ave();//主卷拉力滤波

IF (NOT SaveEngineState) OR (NOT CANI_WorkModeSwitch) THEN 
	//Y71 Y72 Y73不输出
	GVL_SaveEngine.Y72OutPutState:=0;
	GVL_SaveEngine.Y71OutPutState:=0;
	Y73:=0;
	SaveEngineMode:=0;
	control();//不节能
ELSE//打开节能开关，在作业档才进入节能模式(*CANI_WorkModeSwitch=1作业挡情况下*)
	SaveEngineControl();
END_IF

END_PROGRAM

// StandardPLC/Application/SaveEngine/MainWinTension_Ave
PROGRAM MainWinTension_Ave
VAR
	MainWinchTension_Sum:UINT:=0;
	MainWinchTension:ARRAY[0..30] OF UINT;
	m: UINT:=30;	
	MainWinchTension_i:UINT;
END_VAR

//主卷拉力滤波,每循环计算一次前面30个数据的平均值
MainWinchTension_Sum:=0;
MainWinchTension[m]:=CANO_MainWinchTension;
FOR MainWinchTension_i:=0 TO (m-1) BY 1 DO
	MainWinchTension[MainWinchTension_i]:=MainWinchTension[MainWinchTension_i+1];
	MainWinchTension_Sum:=MainWinchTension_Sum+MainWinchTension[MainWinchTension_i];
END_FOR
MainWinchTension_Ave:= (MainWinchTension_Sum)/(m);

END_PROGRAM

// StandardPLC/Application/SaveEngine/SaveEngineControl
PROGRAM SaveEngineControl
VAR
	DI_PWM_JOYX_L: BOOL;
	DI_PWM_JOYY_L: BOOL;
	DI_PWM_JOYX_R: BOOL;
	DI_PWM_JOYY_R: BOOL;
	DI_PWM_JOY_Jiao_R: BOOL;
	DI_PWM_JOY_Jiao_L: BOOL;
	LvZhang_move: BOOL;
	BianFu_move:BOOL;
	JieSuoBool: BOOL;
	TIME_50ms:TON;
	TIME_55ms:TOF;
	TIME_2000ms:TOF;
	start_move: BOOL;
	T1:TIME;
	
	(*节能声明变量*)
	TIME_30ms_DNweidong:TON;//手柄微动计时,600改为30
	DNweidongTimecouter:UINT;
	Timecouter:UINT;
	UPweidongTimecouter:UINT;
	DNFlag_1:BOOL;
	DNTimecouter_1:UINT;	
	DNweidongFlag_0:BOOL;
	DNweidongFlag:BOOL;//微动下放标志
	DownFlag:BOOL;//正常下放标志
	UPweidongFlag_0:BOOL;	
	UPweidongFlag:BOOL;	//微动上提标志
	UPFlag:BOOL;	//正常上提标志
	Energe_NotEnough_Flag:BOOL;//能量不足标志位
	MainWinch_singlmove:BOOL;
    SaveEngineUpFlag:BOOL:=FALSE;//节能上升标志
	SaveEngineTimer100Ms: TON;//节能10ms定时器
	SaveEngineDownFlag:BOOL:=FALSE;//节能下降标志
	SaveEngineDownTimer:UINT:=0;//节能下降计时器
	SaveEngineDownTimer1:UINT:=0;//节能下降计时器1(节能页面刚开始下降，2s内不对flag1to0做判断)
	SaveEngineUpTimer:UINT:=0;//节能上升计时器

	
	falg_1to0: BOOL :=FALSE;
	TIME_1000ms_M2:TON;//M2大于100bar1s
	TIME_100ms_M2:TON;
	TIME_1000ms_M2in:BOOL;
	TIME_100ms_joy:TON;//手柄信号每200ms一次存给中间变量,用于主卷电磁阀主泵卸荷阀赋值

	PWM_JOYY_L_UP_Avrg: UINT;//判断松手柄的中间变量,之前n个平均值
	JoyDesArray:ARRAY [0..10] OF UINT;
	n: UINT:=10;
	JoyDes_i:UINT;
	JoyDes_sum:UINT:=0;
	TIME_1000ms_Desto0:TON;//手柄回位至中位后维持1s
	Mode1_flag:BOOL;
	Mode0_flag:BOOL;
	Mode8_flag:BOOL;
	JoyDesArraymax: UINT;
	JoyDesArraymin: UINT;
	RAMP_joy:RAMP_INT;
	FudongEnable:BOOL;
	CC:UINT;

	TIME_100ms_M2in: BOOL;
	MainWinch_singlmove_1: BOOL;
END_VAR

IF DI_LHandle_SB5 THEN
	DOH_Y59:=TRUE;
ELSE
	DOH_Y59:=FALSE;
END_IF

//延时断电,暂时没有外部电气线路，没启用此功能
TIME_2000ms(IN:=DIH_power3,PT:=T#2S);
IF(TIME_2000ms.Q)THEN
	DOH_YS3:=TRUE;
ELSE
	DOH_YS3:=FALSE;
END_IF
IF DIL_SQ4 THEN//主卷上限位开关触发,需要在调整档工况改变DIL_SQ4
	IF(NOT JieSuoBool) THEN//调整档模式下JieSuoBool才会置true,目前为作业档模式,false
		PWM_JOYY_L_DOWN:=0;
	END_IF
END_IF
//主卷下限位及解锁
//主卷下放限制

IF( CANO_MainWinchTension*100<PAR_MainWinchLaLi_Low) AND (NOT DI_LHandle_SB1) AND (CANI_WorkModeSwitch)THEN
	PWM_JOYY_L_UP:=0;
END_IF



TIME_50ms(in:=start_move,pt:=T1);
TIME_55ms(in:=start_move,pt:=T#500MS);
IF( LeftMove_move OR  RightMove_move  OR   MainWinch_move OR PowerHead_move OR ViceWinch_move )THEN
	start_move:=TRUE;
ELSE
	start_move:=FALSE;
END_IF
IF NOT DIL_SQ3 THEN(*先导控制输入*)
	IF PWM_JOYX_L_UP>10 OR PWM_JOYX_L_DOWN>10 THEN  DI_PWM_JOYX_L := TRUE;ELSE DI_PWM_JOYX_L:=FALSE;END_IF(*左手柄左右动作*)
	IF PWM_JOYY_L_UP>10 OR PWM_JOYY_L_DOWN>10 THEN  DI_PWM_JOYY_L := TRUE;ELSE DI_PWM_JOYY_L:=FALSE;END_IF(*左手柄前后动作*)
	IF PWM_JOYX_R_UP>10 OR PWM_JOYX_R_DOWN>10 THEN  DI_PWM_JOYX_R := TRUE;ELSE DI_PWM_JOYX_R:=FALSE;END_IF(*右手柄左右动作*)
	IF PWM_JOYY_R_UP>10 OR PWM_JOYY_R_DOWN>10 THEN  DI_PWM_JOYY_R := TRUE;ELSE DI_PWM_JOYY_R:=FALSE;END_IF(*右手柄前后动作*)
	IF PWM_JOY_Jiao_L_UP>10 OR PWM_JOY_Jiao_L_DOWN>10 THEN  DI_PWM_JOY_Jiao_L:= TRUE;ELSE DI_PWM_JOY_Jiao_L:=FALSE;END_IF(*左脚踏前后动作*)
	IF PWM_JOY_Jiao_R_UP>10 OR PWM_JOY_Jiao_R_DOWN>10 THEN  DI_PWM_JOY_Jiao_R := TRUE;ELSE DI_PWM_JOY_Jiao_R:=FALSE;END_IF(*左脚踏左右动作*)
ELSE
	DI_PWM_JOYX_L:=FALSE;
	DI_PWM_JOYY_L:=FALSE;
	DI_PWM_JOYX_R:=FALSE;
	DI_PWM_JOYY_R:=FALSE;
	DI_PWM_JOY_Jiao_L:=FALSE;
	DI_PWM_JOY_Jiao_R:=FALSE;
END_IF
(*动作标志*)
IF DI_PWM_JOYY_L THEN MainWinch_move:=TRUE; ELSE MainWinch_move:=FALSE;END_IF(*主卷扬动作*)
IF DI_PWM_JOYX_L THEN Rotation_move:=TRUE; ELSE Rotation_move:=FALSE;END_IF(*回转动作*)
(*IF CANI_WorkModeSwitch THEN   (*作业挡情况下*)*)
	IF DI_PWM_JOYX_R THEN PowerHead_move:=TRUE;ELSE PowerHead_move:=FALSE;END_IF(*动力头回转动作*)
	IF DI_PWM_JOYY_R THEN JiaYa_move:=TRUE;ELSE JiaYa_move:=FALSE;END_IF(*动力头加压动作*)
	LvZhang_move:=FALSE;
	BianFu_move:=FALSE;
	ViceWinch_move:=FALSE;
	LeftMove_move:=FALSE;
	RightMove_move:=FALSE;
	
//先导控制
IF(NOT DIL_SQ3) AND NOT VarGpsSystemLockedState THEN
	DOH_Y51:=TRUE;
ELSE
	DOH_Y51:=FALSE;
END_IF
	

(*模式0不节能模式 /模式1节能下降 /模式2节能上升/模式3上升能量不足/模式4手柄中位模式/模式5泄压模式*)
(*******************模式判断条件输入**************************)
IF (NOT PowerHead_move) AND (NOT Rotation_move) AND (NOT JiaYa_move) AND (NOT DIL_SQ3) THEN//LvZhang_move BianFu_move ViceWinch_move LeftMove_move RightMove_move
	MainWinch_singlmove:=TRUE;
ELSE
	MainWinch_singlmove:=FALSE;
END_IF

IF (NOT PowerHead_move) AND (NOT Rotation_move) AND (NOT DIL_SQ3) THEN//主卷动作和动力头加压情况下  1模式收能
	MainWinch_singlmove_1:=TRUE;
ELSE
	MainWinch_singlmove_1:=FALSE;
END_IF
//微动定时器
TIME_30ms_DNweidong(IN:=NOT TIME_30ms_DNweidong.Q , PT:= T#30MS, Q=> , ET=> );
IF TIME_30ms_DNweidong.Q THEN
	IF DNFlag_1 THEN
		IF DNTimecouter_1<=16#FFFF THEN
				DNTimecouter_1:=DNTimecouter_1+1;
		ELSE
			
				DNTimecouter_1:=16#FFFF;
		END_IF
		
	ELSIF DNweidongFlag_0 THEN
		IF DNweidongTimecouter<=16#FFFF THEN
				DNweidongTimecouter:=DNweidongTimecouter+1;
		ELSE
				DNweidongTimecouter:=16#FFFF;
		END_IF
	ELSIF (UPweidongFlag_0) THEN
		IF UPweidongTimecouter<=16#FFFF THEN
		UPweidongTimecouter:=UPweidongTimecouter+1;
		ELSE
				UPweidongTimecouter:=16#FFFF;
		END_IF
	END_IF	
END_IF
//微动判断
IF (PWM_JOYY_L_UP>10)THEN 
	IF NOT DownFlag THEN
		IF(PWM_JOYY_L_UP<=500) OR DNweidongFlag THEN//之前不是1模式,只要手柄值小于60%
			DNweidongFlag:=TRUE;//4模式进入7模式(进入1模式后退出)
		END_IF
	END_IF
	IF DNweidongFlag THEN
		IF (PWM_JOYY_L_UP<=500) THEN	//7模式进入(或再次进入)1模式定时条件
			DNFlag_1:=FALSE;
			DNTimecouter_1:=0;
		ELSE	
			DNFlag_1:=TRUE;//注释 	直接进入1模式
		END_IF
	END_IF
	IF DNFlag_1 OR DownFlag THEN//7进1模式判断,或再次进入1模式  //这段不要计时 直接进入1模式
		DNweidongFlag:=FALSE;//7模式退出
		DNweidongTimecouter:=0;
		DownFlag:=TRUE;//7进入1模式
		DNFlag_1:=FALSE;
		IF (PWM_JOYY_L_UP<=500) THEN
			DNweidongFlag_0:=TRUE;//1模式进入7模式定时条件
		ELSE
			DNweidongFlag_0:=FALSE;
			DNweidongTimecouter:=0;
		END_IF
	END_IF
	IF (DNweidongTimecouter>=10) THEN
		DNweidongFlag:=TRUE;//1模式进入7模式(上提或中位或再次进入1模式退出)
		DownFlag:=FALSE;//1模式退出
		DNTimecouter_1:=0;
		DNweidongFlag_0:=FALSE;
	END_IF
ELSE
	DNweidongFlag:=FALSE;//上提或中位时7模式退出
	DNFlag_1:=FALSE;
	DNweidongFlag_0:=FALSE;
	DownFlag:=FALSE;
	DNTimecouter_1:=0;
	DNweidongTimecouter:=0;
END_IF
//上提：手柄开度小于60%持续600ms(10个30ms定时器循环),则进入上升微动,不足600ms或其他都正常上提
IF (PWM_JOYY_L_DOWN>10)THEN 
	IF (PWM_JOYY_L_DOWN<500)THEN
		UPweidongFlag_0:=TRUE;
	ELSE
		UPweidongFlag_0:=FALSE;
		UPweidongTimecouter:=0;
	END_IF
	IF (UPweidongTimecouter=10) THEN
		UPweidongFlag:=TRUE;//微动上提
		UPFlag:=FALSE;
		UPweidongFlag_0:=FALSE;
	ELSE
		UPweidongFlag:=FALSE;
		UPFlag:=TRUE;//正常上提
	END_IF
ELSE
	UPweidongTimecouter:=0;
	UPweidongFlag_0:=FALSE;
	UPFlag:=FALSE;	
	UPweidongFlag:=FALSE;
END_IF

SaveEngineTimer100Ms(IN:=(NOT SaveEngineTimer100Ms.Q) , PT:=T#100MS, Q=> , ET=> );

IF(SaveEngineTimer100Ms.Q)THEN
		//下降收满能计时器
	IF SaveEngineDownFlag AND (AI_PAcPre>=300)THEN//Px收能到310开始计时xxms后退出收能
		IF SaveEngineDownTimer<=16#FFFF THEN
			SaveEngineDownTimer:=SaveEngineDownTimer+1;
		ELSE
			SaveEngineDownTimer:=16#FFFF;
		END_IF	
	ELSE
		SaveEngineDownTimer:=0;
	END_IF
		//上升放完能计时器
	IF SaveEngineUpFlag AND (AI_PAcPre<=175)THEN//Px放能到180开始计时xxms后退出放能 180-195
		IF SaveEngineUpTimer<=16#FFFF THEN
			SaveEngineUpTimer:=SaveEngineUpTimer+1;
		ELSE
			SaveEngineUpTimer:=16#FFFF;
		END_IF	
	ELSE
	SaveEngineUpTimer:=0;
	END_IF

  //进入2模式2s计时器
	IF 2=GVL_SaveEngine.SaveEngineMode THEN
		IF Mode2Timer<=16#FFFF THEN
			Mode2Timer:=Mode2Timer+1;
		ELSE
			Mode2Timer:=16#FFFF;
		END_IF	
	ELSE
		Mode2Timer:=0;
	END_IF

  //进入1模式0.5s计时器
	IF 1=GVL_SaveEngine.SaveEngineMode THEN//180改为130
		IF Mode1Timer<=16#FFFF THEN
			Mode1Timer:=Mode1Timer+1;
		ELSE
			Mode1Timer:=16#FFFF;
		END_IF	
	ELSE
	Mode1Timer:=0;
	END_IF

  //进入1模式Y71 Y72开启顺序计时器
	IF 1=GVL_SaveEngine.SaveEngineMode THEN//180改为130
		IF Mode1Timer_1<=16#FFFF THEN
			Mode1Timer_1:=Mode1Timer_1+1;
		ELSE
			Mode1Timer_1:=16#FFFF;
		END_IF	
	ELSE
	Mode1Timer_1:=0;
	END_IF
	
	//进入4模式计时器,没有用到
	IF 4=GVL_SaveEngine.SaveEngineMode THEN//180改为130
		IF Mode4Timer<=16#FFFF THEN
			Mode4Timer:=Mode4Timer+1;
		ELSE
			Mode4Timer:=16#FFFF;
		END_IF		
	ELSE
			Mode4Timer:=0;
	END_IF
	//进入7模式Y71 Y72关闭顺序计时器
	IF 7=GVL_SaveEngine.SaveEngineMode THEN//180改为130
		IF Mode7Timer<=16#FFFF THEN
			Mode7Timer:=Mode7Timer+1;
		ELSE
			Mode7Timer:=16#FFFF;
		END_IF		
	ELSE
			Mode7Timer:=0;
	END_IF

	
	//进入8模式Y71 Y72关闭顺序计时器	
	IF 8=GVL_SaveEngine.SaveEngineMode THEN//180改为130
		IF Mode8Timer<=16#FFFF THEN
			Mode8Timer:=Mode8Timer+1;
		ELSE
			Mode8Timer:=16#FFFF;
		END_IF		
	ELSE
			Mode8Timer:=0;
	END_IF
	//进入10模式Y71 Y72关闭顺序计时器
	IF 10=GVL_SaveEngine.SaveEngineMode THEN//180改为130
		IF Mode10Timer<=16#FFFF THEN
			Mode10Timer:=Mode10Timer+1;
		ELSE
			Mode10Timer:=16#FFFF;
		END_IF		
	ELSE
			Mode10Timer:=0;
	END_IF
	
	//进入11模式Y71 Y72关闭顺序计时器
	IF 11=GVL_SaveEngine.SaveEngineMode THEN//180改为130
		IF Mode11Timer<=16#FFFF THEN
			Mode11Timer:=Mode11Timer+1;
		ELSE
			Mode11Timer:=16#FFFF;
		END_IF		
	ELSE
			Mode11Timer:=0;
	END_IF
	//进入12模式Y71 Y72关闭顺序计时器
	IF 12=GVL_SaveEngine.SaveEngineMode THEN//180改为130
		IF Mode12Timer<=16#FFFF THEN
			Mode12Timer:=Mode12Timer+1;
		ELSE
			Mode12Timer:=16#FFFF;
		END_IF		
	ELSE
			Mode12Timer:=0;
	END_IF
	
	//手柄回位动作计时器
	IF JoyDesFlag THEN
		IF JoyDesTimer<=16#FFFF THEN
			JoyDesTimer:=JoyDesTimer+1;
		ELSE
			JoyDesTimer:=16#FFFF;
		END_IF
	ELSE
		JoyDesTimer:=0;
	END_IF

	
END_IF
//M2压力高计时 M2>140 持续400ms 马达排量已降到最小 前一个模式是1模式则退出收能切到11模式
IF ((GVL_SaveEngine.AI_PM2Pre>=150)) THEN//100改为140  300->140—>150
	TIME_1000ms_M2in:=TRUE;
ELSE
	TIME_1000ms_M2in:=FALSE;
END_IF
TIME_1000ms_M2(IN:=TIME_1000ms_M2in , PT:= T#500MS );//400-500
IF (TIME_1000ms_M2.Q AND (GVL_SaveEngine.PWM_Y33_SET_Target>=465) AND (1=GVL_SaveEngine.SaveEngineMode)) THEN
	falg_1to0:=TRUE;
END_IF
//M2压力>140 持续100ms计时器  没有用到

IF ((GVL_SaveEngine.AI_PM2Pre>=140)) THEN//100改为140  300->140—>150
	TIME_100ms_M2in:=TRUE;
ELSE
	TIME_100ms_M2in:=FALSE;
END_IF
(*
TIME_100ms_M2(IN:=TIME_100ms_M2in , PT:= T#100MS );
IF (TIME_100ms_M2.Q AND GVL_SaveEngine.PWM_Y33_SET_Target>=450 AND  (1=GVL_SaveEngine.SaveEngineMode)) THEN
	M2_Press_H_C:=TRUE;
END_IF
*)

(*
IF ((GVL_SaveEngine.AI_PM2Pre>=140)) THEN//100改为140  300->140—>150
	TIME_100ms_M2in:=TRUE;
ELSE
	TIME_100ms_M2in:=FALSE;
END_IF
TIME_100ms_M2(IN:=TIME_100ms_M2in , PT:= T#100MS );
IF (TIME_100ms_M2.Q AND GVL_SaveEngine.PWM_Y33_SET_Target>=450 AND  (1=GVL_SaveEngine.SaveEngineMode)) THEN
	M2_Press_H_C:=TRUE;
END_IF
*)

//左手柄Y方向回位过程,用于减缓手柄信号斜坡的中间变量，弃用
RAMP_joy(
	IN:= UINT_TO_INT(PWM_JOYY_L_UP), 
	ASCEND:= 200, 
	DESCEND:=15, 
	TIMEBASE:=T#500MS , 
	RESET:= FALSE, 
	OUT=>PWM_JOYY_L_UP_1);
	
PWM_JOYY_L_UP_1:=LIMIT(0,PWM_JOYY_L_UP_1,1000);

//左手柄Y方向回收动作判断
JoyDes_sum:=0;
JoyDesArray[n]:=PWM_JOYY_L_UP;
	//滤波
FOR JoyDes_i:=0 TO (n-1) BY 1 DO
	JoyDesArray[JoyDes_i]:=JoyDesArray[JoyDes_i+1];
	JoyDes_sum:=JoyDes_sum+JoyDesArray[JoyDes_i];
	PWM_JOYY_L_UP_Avrg:= (JoyDes_sum)/(n);
END_FOR
IF (PWM_JOYY_L_UP_Avrg>PWM_JOYY_L_UP) THEN
	JoyDesFlag:=TRUE;
ELSE
	JoyDesFlag:=FALSE;	
END_IF
//回中位标志,1s后标志位清0，即12模式进入后会维持12模式1s
IF (JoyDesFlag)AND (PWM_JOYY_L_UP<10) THEN
	JoyDesto0_flag:=TRUE;
END_IF
TIME_1000ms_Desto0(IN:=JoyDesto0_flag, PT:=T#1000MS );
IF(TIME_1000ms_Desto0.Q) THEN
	JoyDesto0_flag:=FALSE;	
END_IF

//Tension_Ton1(IN:=(CANO_MainWinchTension>90),PT:=T#500MS);
(*连续20个值*)
(*
MainWinchTension_Count:=MainWinchTension_Count+1;

IF MainWinchTension_Count=21 THEN
	MainWinchTension_Ave:= MainWinchTension_Sum/20;
	MainWinchTension_Count:=0;
	MainWinchTension_Sum:=0;
ELSE
	MainWinchTension_Sum:=CANO_MainWinchTension+MainWinchTension_Sum;
END_IF
*)

(*******************模式判断**************************)
IF GVL_SaveEngine.AcDecompression THEN
	SaveEngineMode:=5;//泄压模式
	FudongEnable:=FALSE;
ELSE
	FudongEnable:=TRUE;
	IF EngineSpeedTarget<1300 THEN
		GVL_SaveEngine.SaveEngineMode:=9;
	ELSE
		IF JoyDesto0_flag AND Mode1_flag THEN
			GVL_SaveEngine.SaveEngineMode:=12;//节能下放回至中位模式,优先级高于其他模式
			M2_Press_H_C:=FALSE;
			falg_1to0:=FALSE;
		ELSE
			IF MainWinch_singlmove AND (UPFlag)THEN //上提 
				Mode0_flag:=FALSE;
				Mode8_flag:=FALSE;
				Mode1_flag:=FALSE;
				SaveEngineDownFlag:=FALSE;
				//放能条件修改 大于标定值多少合适？
				IF ((AI_PAcPre>220 AND MainWinchTension_Ave>(Max_MainWinchTension-15)) OR (AI_PAcPre<=220 AND MainWinchTension_Ave>(Max_MainWinchTension-15)) OR SaveEngineUpFlag) AND NOT Energe_NotEnough_Flag THEN //155->195 195->200
				//IF ((AI_PAcPre>220 AND MainWinchTension_Ave>125) OR (AI_PAcPre<=220 AND MainWinchTension_Ave>110)) OR SaveEngineUpFlag) AND NOT Energe_NotEnough_Flag THEN //155->195 195->200
					SaveEngineUpFlag:=TRUE;
					SaveEngineMode:=2;//节能上升模式
					IF SaveEngineUpTimer>=1 THEN//如果蓄能器油压小于等于180bar并持续200ms切到上升能量不足模式
					SaveEngineUpFlag:=FALSE;
					Energe_NotEnough_Flag:=TRUE;
					SaveEngineMode:=3;//上升能量不足模式
					END_IF  
				ELSE				
					SaveEngineMode:=3;//上升能量不足模式
				END_IF
			ELSIF MainWinch_singlmove AND (UPweidongFlag) THEN //微动上升 
				Mode0_flag:=FALSE;
				Mode8_flag:=FALSE;
				Mode1_flag:=FALSE;
				SaveEngineMode:=6;//上升微动模式
				SaveEngineDownFlag:=FALSE;
			//下放	
			ELSIF MainWinch_singlmove_1 AND (DownFlag)THEN //下放 
				SaveEngineUpFlag:=FALSE;
				Mode0_flag:=FALSE;
				Energe_NotEnough_Flag:=FALSE;
				IF(AI_PAcPre<280) OR SaveEngineDownFlag THEN //蓄能器油压小于280bar收能
					SaveEngineDownFlag:=TRUE;
					IF (falg_1to0) THEN//如果M2压力高于14mpa
						GVL_SaveEngine.SaveEngineMode:=11;//下放进口压力高模式
						M2_Press_H_C:=FALSE;
						Mode1_flag:=FALSE;
					ELSIF (SaveEngineDownTimer>=2) OR Mode8_flag THEN//如果蓄能器油压大于等于280bar并持续200ms结束收能  
							GVL_SaveEngine.SaveEngineMode:=8;//下放收满能模式
							Mode8_flag:=TRUE;
							Mode1_flag:=FALSE;
					ELSE				
							GVL_SaveEngine.SaveEngineMode:=1;//节能下降模式
							Mode1_flag:=TRUE;
							Mode8_flag:=FALSE;
					END_IF
				ELSE  
					GVL_SaveEngine.SaveEngineMode:=10;//下放能量过高模式
					Mode1_flag:=FALSE;
					Mode8_flag:=FALSE;
				END_IF
				
			ELSIF MainWinch_singlmove AND  (DNweidongFlag) THEN //微动下放 
				SaveEngineMode:=7;//下放微动模式
				SaveEngineUpFlag:=FALSE;
				Mode1_flag:=FALSE;
				Mode0_flag:=FALSE;
				Mode8_flag:=FALSE;
				Energe_NotEnough_Flag:=FALSE;
			//中位
			ELSIF MainWinch_singlmove AND ( PWM_JOYY_L_UP<=10) AND (PWM_JOYY_L_DOWN<=10) AND (NOT Mode0_flag )THEN	
					falg_1to0:=FALSE;
					Mode8_flag:=FALSE;
					SaveEngineUpFlag:=FALSE;
					SaveEngineDownFlag:=FALSE;
					GVL_SaveEngine.SaveEngineMode:=4;//手柄中位模式
					M2_Press_H_C:=FALSE;
					Energe_NotEnough_Flag:=FALSE;
			ELSE
			falg_1to0:=FALSE;
			Mode1_flag:=FALSE;
			Mode0_flag:=TRUE;
			Mode8_flag:=FALSE;
			Energe_NotEnough_Flag:=FALSE;//不节能标志位置false
			GVL_SaveEngine.SaveEngineMode:=9;//不节能模式
			END_IF
		END_IF
	END_IF
END_IF
(*******************节能控制阀主阀主泵输出执行**************************)
IF(GVL_SaveEngine.SaveEngineMode=1)THEN//节能下降模式
	SaveEngineMode_1();
ELSIF(GVL_SaveEngine.SaveEngineMode=2)THEN//节能上升模式
	SaveEngineMode_2();
ELSIF(GVL_SaveEngine.SaveEngineMode=3)THEN//上升能量不足模式
	SaveEngineMode_3();
ELSIF(GVL_SaveEngine.SaveEngineMode=4)THEN//手柄中位模式
	SaveEngineMode_4();
ELSIF(GVL_SaveEngine.SaveEngineMode=5)THEN//泄压模式
	SaveEngineMode_5();
ELSIF(GVL_SaveEngine.SaveEngineMode=6)THEN//上升微动模式
	SaveEngineMode_6();
ELSIF(GVL_SaveEngine.SaveEngineMode=7)THEN//下放微动模式
	SaveEngineMode_7();
ELSIF(GVL_SaveEngine.SaveEngineMode=8)THEN//下放收满能模式
	SaveEngineMode_8();
ELSIF(GVL_SaveEngine.SaveEngineMode=10)THEN//下放能量过高模式
	SaveEngineMode_10();
ELSIF(GVL_SaveEngine.SaveEngineMode=11)THEN//下放进口压力高模式
	SaveEngineMode_11();
ELSIF(GVL_SaveEngine.SaveEngineMode=12)THEN//节能下降回至中位模式,
	SaveEngineMode_12();
//	SaveEngineMode_4();
ELSIF(GVL_SaveEngine.SaveEngineMode=9)THEN//不节能模式,
	SaveEngineMode_9();
	//control();
ELSE
	//control();
	SaveEngineMode_9();
END_IF

	(*冷却风扇控制*)
	IF NOT CANI_ColdFunSwitch  THEN
		IF(CANO_Hyd_Tem>60)THEN
			PWM_Y49_SET := PAR_ValveD_NegFull;
		END_IF
		
		IF(CANO_Hyd_Tem<60)THEN
			PWM_Y49_SET := 0;		
		END_IF
	ELSE
		PWM_Y49_SET := PAR_ValveD_NegFull;
	END_IF
	
	(*主卷浮动*)
	IF FudongEnable AND ((DIH_SA8 OR DI_LHandle_SB3 OR CANI_Button_FloatSwitch) AND CANI_MaiWinFloatSwitch AND (NOT DIL_SQ3)) THEN
		DOH_Y55:=TRUE;
		DOH_Y56:=TRUE;
		DOH_Y64:=TRUE;
		GVL_SaveEngine.Y74:=TRUE;
		GVL_SaveEngine.Y72OutPutState:=0;
		GVL_SaveEngine.Y71OutPutState:=0;
		Y73:=0;
	ELSE
		IF (GVL_SaveEngine.AcDecompression) THEN
			DOH_Y56:=TRUE;			
			IF AI_PAcPre<=150 THEN
				DOH_Y64:=FALSE;
				GVL_SaveEngine.Y74:=FALSE;
			END_IF
		ELSE
			DOH_Y56:=FALSE;			
		END_IF
		DOH_Y55:=FALSE;
		//GVL_SaveEngine.Y74:=FALSE;
	END_IF

	//主卷动作及浮动时开锁
IF  MainWinch_move OR DOH_Y55 THEN
	DOH_Y53 := TRUE;
	DOH_Y64:=TRUE;
	GVL_SaveEngine.Y74:=TRUE;
ELSE
	DOH_Y53 := FALSE;	
	DOH_Y64:=FALSE;
	GVL_SaveEngine.Y74:=FALSE;
END_IF
	
	IF(UIGroupVoltage0<2000 OR UIGroupVoltage1<2000 OR UIGroupVoltage2<2000 
	   OR UIGroupVoltage3<2000 OR UIGroupVoltage4<2000 OR UIGroupVoltage5<2000) THEN
		reset111:=TRUE;
	ELSE
		reset111:=FALSE;
	END_IF

END_PROGRAM

// StandardPLC/Application/SaveEngine/SaveEngineMode_1
PROGRAM SaveEngineMode_1
VAR
	PWM_Y1_Target_1: UINT;//1 节能下降缓冲 
	PWM_Y2_Target_1: UINT;//1
	PWM_Y1_Target_2: UINT;//1 
	PWM_Y2_Target_2: UINT;//1 
	JianGEse:REAL:=2;//1
	QPump:REAL;//1 匹配的下降主泵排量计算
	PumpDispl:REAL ;//1 匹配的下降主泵排量计算
	RopeSpeedMax :REAL;//1 最大下放速度,m/min
	RopeSpeedTarget :REAL;//1 目标下放速度
	WinchSpeedTarget :REAL;//1 卷扬马达速度,r/min
	WinchDisplTarget:REAL:=216;//1 主卷排量,ml/r
	QMotorTarget :REAL :=0;//1 马达需求流量	,
	PAR_Y1_PosFull:UINT:=600;
	PAR_Y2_PosFull:UINT:=600;
	Time_1s:TON;
	Time_1_1s:TON;
	Mod1CasePWM_Y1:UINT;
	PWM_Y12_SET_Tatget: UINT;
	PWM_Y11_SET_Tatget: UINT;
	Timer_1s: BOOL;
	Y73_Flag: BOOL;
	Flag_M:BOOL;
	TON1:TON;
	TON2:TON;
	TON3:TON;
	AI_PM2Pre_Flag:BOOL;
	AI_PM2Pre_Flag1:BOOL;
	AI_PM2Pre_Flag2:BOOL;
	AI_PM2Pre_Flag3:BOOL;
	PM2Pre_Rtrig:R_TRIG;
	PM2Pre_Rtrig1:R_TRIG;
	PM2Pre_Rtrig2:R_TRIG;
	PM2Pre_Rtrig3:R_TRIG;
	A:UINT:=1;
	B:UINT:=1;
	Mod1CasePWM_Y11:UINT;
	PWM_Y23_SET_Taget: UINT;
	PWM_Y24_SET_Taget: UINT;
	
	RAMP22:RAMP_INT;
	RAMP23:RAMP_INT;
	RAMP24:RAMP_INT;
	PWM_Y23_SET_Taget1:INT;
	PWM_Y24_SET_Taget1:INT;
	PWM_Y18_SET_Taget1:INT;
	PWM_Y18_SET_Taget:UINT;
	ASCEND_value2:INT;
	ASCEND_value:INT;
	
END_VAR

(*******************节能控制阀主阀主泵输出执行**************************)
//节能下降	
	(****错开Y71和Y72的开启时间 降低微开到1模式M1压力****)
	(*IF Mode1Timer_1>2 THEN
		//GVL_SaveEngine.Y72OutPutState:=1;
		GVL_SaveEngine.Y71OutPutState:=1;
	END_IF

	IF Mode1Timer_1>3 THEN
		GVL_SaveEngine.Y72OutPutState:=1;
	END_IF*)
	
	GVL_SaveEngine.Y71OutPutState:=1;
	GVL_SaveEngine.Y72OutPutState:=1;
	DOH_Y56:=FALSE;
	//开Y73补油条件：1、回手柄持续100ms且手柄开度<70%   2、M2<30开启Y73至M2>45关闭
	IF ((JoyDesFlag)AND(PWM_JOYY_L_UP<700) AND (JoyDesTimer>=1)) THEN
	Y73:=TRUE;
	ELSE
	Y73:=FALSE;	
	END_IF

	IF GVL_SaveEngine.AI_PM2Pre<30 OR Y73_Flag THEN
		Y73:=TRUE;
		Y73_Flag:=TRUE;
	END_IF
	IF GVL_SaveEngine.AI_PM2Pre>45 THEN
		Y73:=FALSE;
		Y73_FLag:=FALSE;
	END_IF
//M2>6MPa,每过1s Y33+18,排量减10，至Y33>450,之后若M2压力高于14MPa持续1s，切出1模式进入11模式(在外层实现模式切换)
(*
IF (GVL_SaveEngine.AI_PM2Pre>=50) THEN  
		IF (GVL_SaveEngine.AI_PM2Pre>=100) AND PWM_Y33_SET_Target=450 THEN
			Time_1s(IN:=NOT Time_1s.Q, PT:= T#1S , Q=> , ET=> );	
			IF Time_1s.Q THEN
			GVL_SaveEngine.PWM_Y33_SET_Target:=GVL_SaveEngine.PWM_Y33_SET_Target+18;
			END_IF
		ELSIF (GVL_SaveEngine.PWM_Y33_SET_Target<450) THEN  
			Time_1s(IN:=NOT Time_1s.Q, PT:= T#1S , Q=> , ET=> );	
			IF Time_1s.Q THEN
			GVL_SaveEngine.PWM_Y33_SET_Target:=GVL_SaveEngine.PWM_Y33_SET_Target+18;//1s排量减10，
			END_IF	
		ELSIF(GVL_SaveEngine.PWM_Y33_SET_Target>450) AND GVL_SaveEngine.AI_PM2Pre<100 THEN
			Time_1s(IN:=NOT Time_1s.Q, PT:= T#1S , Q=> , ET=> );	
			IF Time_1s.Q THEN
			GVL_SaveEngine.PWM_Y33_SET_Target:=GVL_SaveEngine.PWM_Y33_SET_Target-18;
			END_IF
		END_IF
ELSIF (GVL_SaveEngine.AI_PM2Pre<=30) THEN
		IF (GVL_SaveEngine.PWM_Y33_SET_Target>=230) THEN
			Time_1_1s(IN:=NOT Time_1_1s.Q, PT:= T#200MS , Q=> , ET=> );	
			IF Time_1_1s.Q THEN
			GVL_SaveEngine.PWM_Y33_SET_Target:=GVL_SaveEngine.PWM_Y33_SET_Target-18;//1s排量加10，
			END_IF
		END_IF				
END_IF

	PWM_Y33_SET := LIMIT(378,GVL_SaveEngine.PWM_Y33_SET_Target,468);//去掉原有坡度执行防止干扰
*)	
	
	TON1(IN:=NOT TON1.Q AND GVL_SaveEngine.AI_PM2Pre<30 ,PT:=T#200MS);
	TON2(IN:=NOT TON2.Q AND GVL_SaveEngine.AI_PM2Pre>=50 ,PT:=T#500MS);
	IF TON2.Q AND GVL_SaveEngine.PWM_Y33_SET_Target<500 THEN
		AI_PM2Pre_Flag1:=TRUE;
	ELSE
		AI_PM2Pre_Flag1:=FALSE;
	END_IF
	IF GVL_SaveEngine.PWM_Y33_SET_Target>=230 AND TON1.Q  THEN
		AI_PM2Pre_Flag3:=TRUE;
	ELSE
		AI_PM2Pre_Flag3:=FALSE;
	END_IF

	PM2Pre_Rtrig1(CLK:=AI_PM2Pre_Flag1);
	PM2Pre_Rtrig3(CLK:=AI_PM2Pre_Flag3);

	IF(PM2Pre_Rtrig1.Q)THEN
		A:=A+1;
		GVL_SaveEngine.PWM_Y33_SET_Target:=GVL_SaveEngine.PWM_Y33_SET_Target+17;
		AI_PM2Pre_Flag1:=FALSE;
	END_IF
	
	IF(PM2Pre_Rtrig3.Q)THEN
		B:=B+1;
		GVL_SaveEngine.PWM_Y33_SET_Target:=GVL_SaveEngine.PWM_Y33_SET_Target-17;
		AI_PM2Pre_Flag3:=FALSE;
	END_IF
	//目标排量范围限制在80-110
	GVL_SaveEngine.PWM_Y33_SET_Target:=LIMIT(417,GVL_SaveEngine.PWM_Y33_SET_Target,465);//396-378  下降初始排量120cc/r  0423  120 396 0427
	PWM_Y33_SET := GVL_SaveEngine.PWM_Y33_SET_Target;//去掉原有坡度执行防止干扰
	
	
	IF DIL_SQ3 THEN
		PWM_Y33_SET:=0;
	END_IF														

	(*CASE AI_ECM2_Flag OF
		1: Mod1CasePWM_Y1:=REAL_TO_UINT(362.5+47.8*30/1100*(600-PWM_Y33_SET)/1.85)+40;
		2: Mod1CasePWM_Y1:=REAL_TO_UINT(362.5+47.8*42/1200*(600-PWM_Y33_SET)/1.85)+40;
		3: Mod1CasePWM_Y1:=REAL_TO_UINT(362.5+47.8*55/1450*(600-PWM_Y33_SET)/1.85)+40;
		4: Mod1CasePWM_Y1:=REAL_TO_UINT(362.5+47.8*62/1500*(600-PWM_Y33_SET)/1.85)+40;//调速 //+40
		5: Mod1CasePWM_Y1:=REAL_TO_UINT(362.5+47.8*68/1500*(600-PWM_Y33_SET)/1.85)+0;//
		6: Mod1CasePWM_Y1:=REAL_TO_UINT(362.5+47.8*72/1500*(600-PWM_Y33_SET)/1.85)-20;//
	END_CASE
	*)
	
	
	CASE AI_ECM2_Flag OF
		1: Mod1CasePWM_Y1:=REAL_TO_UINT(362.5+47.8*30/1100*(600-PWM_Y33_SET)/1.85)+40;
		2: Mod1CasePWM_Y1:=REAL_TO_UINT(362.5+47.8*42/1200*(600-PWM_Y33_SET)/1.85)+40;
		3: Mod1CasePWM_Y1:=REAL_TO_UINT(362.5+47.8*55/1450*(600-PWM_Y33_SET)/1.85)+40;
		4: Mod1CasePWM_Y1:=REAL_TO_UINT(362.5+47.8*62/1500*(600-PWM_Y33_SET)/1.85)+120;//40-60
		5: Mod1CasePWM_Y1:=REAL_TO_UINT(362.5+47.8*68/1500*(600-PWM_Y33_SET)/1.85)+120;//0-60
		6: Mod1CasePWM_Y1:=REAL_TO_UINT(362.5+47.8*72/1500*(600-PWM_Y33_SET)/1.85)+120;//-20-60
	END_CASE
	
	(* IF M2_Press_H_C THEN
				Mod1CasePWM_Y1:=REAL_TO_UINT(362.5+47.8*62/1500*(600-PWM_Y33_SET)/1.85)+55;
			ELSE
				Mod1CasePWM_Y1:=REAL_TO_UINT(362.5+47.8*62/1500*(600-PWM_Y33_SET)/1.85)+40;
			END_IF
			*)
	//进入1模式后的前1s限制主泵最大电流
	IF Mode1Timer<=5 THEN 
		CASE SPEED_CASE OF
			1: Mod1CasePWM_Y1:=REAL_TO_UINT(362.5+47.8*30/1100*(600-PWM_Y33_SET)/1.85)+20;//0.5-1
			2: Mod1CasePWM_Y1:=REAL_TO_UINT(362.5+47.8*42/1200*(600-PWM_Y33_SET)/1.85)+20;//0.5-1
			3: Mod1CasePWM_Y1:=REAL_TO_UINT(362.5+47.8*55/1450*(600-PWM_Y33_SET)/1.85)+20 ;
			4: Mod1CasePWM_Y1:=REAL_TO_UINT(362.5+47.8*62/1500*(600-PWM_Y33_SET)/1.85)+20 ;
			5: Mod1CasePWM_Y1:=REAL_TO_UINT(362.5+47.8*68/1500*(600-PWM_Y33_SET)/1.85)+20 ;
			6: Mod1CasePWM_Y1:=REAL_TO_UINT(362.5+47.8*72/1500*(600-PWM_Y33_SET)/1.85)+20 ;
		END_CASE
	END_IF

	
	PWM_Y1_Target:=REAL_TO_UINT(UINT_TO_REAL(PWM_JOYY_L_UP)/1000*(Mod1CasePWM_Y1-PAR_Y1_NegFull)+PAR_Y1_NegFull);
	PWM_Y2_Target:=REAL_TO_UINT(UINT_TO_REAL(PWM_JOYY_L_UP)/1000*(Mod1CasePWM_Y1-PAR_Y2_NegFull)+PAR_Y2_NegFull);

	IF PWM_Y1_Target>700 THEN 
		PWM_Y1_Target:=700;
	END_IF
	IF PWM_Y2_Target>700 THEN 
		PWM_Y2_Target:=700;
	END_IF

(*主泵功率控制*)//1模式去掉了压力波动降低主泵电流的功率控制，只保留了斜坡控制

//区分发动机转速
MainPump_Pressure_Taget1450:=PAR_NegFull_x;
MainPump_Pressure_Taget1600:=PAR_PosFull_x;
MainPump_Pressure_Taget1750:=PAR_Zero_x;

IF EngineSpeedTarget<=1080 THEN SPEED_CASE:=1;
ELSIF EngineSpeedTarget>1080 AND EngineSpeedTarget<=1300 THEN SPEED_CASE:=2;
ELSIF EngineSpeedTarget>1300 AND EngineSpeedTarget<=1520 THEN SPEED_CASE:=3;
ELSIF EngineSpeedTarget>1520 AND EngineSpeedTarget<=1680 THEN SPEED_CASE:=4;
ELSIF EngineSpeedTarget>1680 AND EngineSpeedTarget<=1820 THEN SPEED_CASE:=5;
ELSIF EngineSpeedTarget>1820 THEN SPEED_CASE:=6;;END_IF
//不同转速下的发动机最大功率*)
CASE SPEED_CASE OF
1:  Enginer_Power:=135;
2:  Enginer_Power:=174;
3:  Enginer_Power:=200;
4:  Enginer_Power:=230;
5:  Enginer_Power:=250;
6:  Enginer_Power:=261;
END_CASE
//不同转速下的压力值
IF(CANO_Fubeng_Press>100)THEN
	CASE SPEED_CASE OF
	1:MainPump_Pressure_Taget:=MainPump_Pressure_Taget1000-HELIU_Press_Target1000;
	2:MainPump_Pressure_Taget:=MainPump_Pressure_Taget1200-HELIU_Press_Target1200;
	3:MainPump_Pressure_Taget:=MainPump_Pressure_Taget1450-HELIU_Press_Target1400;
	4:MainPump_Pressure_Taget:=MainPump_Pressure_Taget1600-HELIU_Press_Target1600;
	5:MainPump_Pressure_Taget:=MainPump_Pressure_Taget1750-HELIU_Press_Target1800;
	6:MainPump_Pressure_Taget:=MainPump_Pressure_Taget1900-HELIU_Press_Target1900;
	END_CASE
ELSE
	CASE SPEED_CASE OF
	1:MainPump_Pressure_Taget:=MainPump_Pressure_Taget1000;
	2:MainPump_Pressure_Taget:=MainPump_Pressure_Taget1200;
	3:MainPump_Pressure_Taget:=MainPump_Pressure_Taget1450;
	4:MainPump_Pressure_Taget:=MainPump_Pressure_Taget1600;
	5:MainPump_Pressure_Taget:=MainPump_Pressure_Taget1750;
	6:MainPump_Pressure_Taget:=MainPump_Pressure_Taget1900;
	END_CASE		
END_IF

IF( CANI_ECOSwitch) THEN
	CASE SPEED_CASE OF
	1:MainPump_Pressure_Taget:=MainPump_Pressure_Taget1000-ECO_Press_Target1000;
	2:MainPump_Pressure_Taget:=MainPump_Pressure_Taget1200-ECO_Press_Target1200;
	3:MainPump_Pressure_Taget:=MainPump_Pressure_Taget1450-ECO_Press_Target1400;
	4:MainPump_Pressure_Taget:=MainPump_Pressure_Taget1600-ECO_Press_Target1600;
	5:MainPump_Pressure_Taget:=MainPump_Pressure_Taget1750-ECO_Press_Target1800;
	6:MainPump_Pressure_Taget:=MainPump_Pressure_Taget1900-ECO_Press_Target1900;
	END_CASE
END_IF
MainPump_Pressure:=CANO_MainPUMP_Press1+CANO_MainPUMP_Press2;
//消除滤波
MainPump_Pressure_Subtract:= UINT_TO_INT(MainPump_Pressure-MainPump_Pressure_last1);


//大范围波动
IF MainPump_Pressure_Subtract>270 OR MainPump_Pressure_Subtract<-270 THEN
	Subtract:=TRUE;
ELSE
	Subtract:=FALSE;	
END_IF
	TIME_LvBo4(IN:=Subtract,PT:=T#10MS);
	
IF(TIME_LvBo4.Q) AND (CANO_MainPUMP_Press1>210) THEN 
		MainPump_Pressure_ChangeBool1:=TRUE;
END_IF
	TIME_LvBo1(IN:=MainPump_Pressure_ChangeBool1,PT:=T#2S);
IF(TIME_LvBo1.Q) THEN
	MainPump_Pressure_ChangeBool1 :=FALSE;
END_IF

IF(MainPump_Pressure_ChangeBool1) AND (MainPump_Pressure>MainPump_Pressure_last1) THEN 
	MainPump_Pressure_last1:=MainPump_Pressure;
END_IF

//小范围波动
t_powertime:=TO_TIME(PAR_DeadBand_x);
IF (NOT MainPump_Pressure_ChangeBool1) THEN
	IF(MainPump_Pressure_Subtract>40 OR MainPump_Pressure_Subtract<-40)THEN 
		MainPump_Pressure_ChangeBool:=TRUE;
	ELSE
		MainPump_Pressure_ChangeBool:=FALSE;
	END_IF

	TIME_LvBo2(IN:=MainPump_Pressure_ChangeBool,PT:=t_powertime);//2s-10ms
	IF(TIME_LvBo2.Q )THEN
		MainPump_Pressure_last1:=MainPump_Pressure;
	END_IF	
END_IF


IF PowerHead_move AND NOT(MainWinch_move) THEN
		JianGE2:=0.005;
ELSE
	IF(EngineSpeedTarget>1000 AND EngineSpeedTarget<1300)THEN
		JianGE2:=0.005;
	ELSE
		JianGE2:=0.005;
	END_IF
END_IF
//主泵斜坡的输入=目标值,
	PWM_Y1_Target_OutPut:=PWM_Y1_Target;
	PWM_Y2_Target_OutPut:=PWM_Y2_Target;

IF(EngineSpeedTarget>CANO_SPEED AND CANO_SPEED>400)THEN
	EngineSpeedSub:=EngineSpeedTarget - CANO_SPEED;
ELSE
	EngineSpeedSub:=0;
END_IF

IF(PWM_Y1_Target_OutPut<300)THEN PWM_Y1_Target_OutPut:=300;END_IF	
IF(PWM_Y2_Target_OutPut<300)THEN PWM_Y2_Target_OutPut:=300;END_IF

RAMP15_IN:=PWM_Y1_Target_OutPut;
RAMP16_IN:=PWM_Y2_Target_OutPut;
(*
(******斜坡增步长300 斜坡降步长300->400*****)	
RAMP15(
	IN:=UINT_TO_INT(RAMP15_IN), 
	ASCEND:= 300, 
	DESCEND:= 400, 
	TIMEBASE:=T#1000MS , 
	RESET:=FALSE , 
	OUT=>(PWM_Y1_SET));
(******减斜坡300->400*****)	
RAMP16(
	IN:=UINT_TO_INT(RAMP16_IN), 
	ASCEND:= 300, 
	DESCEND:= 400, 
	TIMEBASE:=T#1000MS , 
	RESET:=FALSE , 
	OUT=>(PWM_Y2_SET));
*)	
	
(*	
	F_RAMP_pump:=1000;  //再快一点  1500  发动机转速掉
	R_RAMP_pump:=300;//6档300  5档250  4 180 3档          2档150  1档100
	
END_IF

RAMP15(
	IN:=UINT_TO_INT(RAMP15_IN), 
	ASCEND:= R_RAMP_pump, 
	DESCEND:= F_RAMP_pump, 
	TIMEBASE:=TIMEBASE_pump , 
	RESET:=FALSE , 
	OUT=>(PWM_Y1_SET));*)
	//主泵电流斜坡根据加压动作和加压压力发生变化
(*   
//主泵电流斜坡给定值 全部变小  防止重载时突然加载时掉速熄火 
CASE AI_ECM2_Flag OF
		1: R_RAMP_pump:=100;
		2: R_RAMP_pump:=150;
		3: R_RAMP_pump:=150;
		4: R_RAMP_pump:=180;
		5: R_RAMP_pump:=250;
		6: R_RAMP_pump:=300;//
END_CASE
*)
       CASE AI_ECM2_Flag OF
                1:F_RAMP_pump:=1500; R_RAMP_pump:=100;                  
                2: 		IF MainWinch_move AND (JiaYa_move OR CANO_JiayaPressure>80)  THEN    //3泵同时起压时，降低主泵的加载速度，避免掉速熄火
                                F_RAMP_pump:=1500; R_RAMP_pump:=100;
                        ELSE
                                F_RAMP_pump:=1500; R_RAMP_pump:=100;//从200降
                                IF  PWM_JOYY_L_UP>10 THEN
                                 F_RAMP_pump:=1500; R_RAMP_pump:=200;
                                END_IF
                        END_IF            
                3:
                        IF MainWinch_move AND (JiaYa_move OR CANO_JiayaPressure>80)  THEN    //3泵同时起压时，降低主泵的加载速度，避免掉速熄火
                                F_RAMP_pump:=1500; R_RAMP_pump:=150;
                        ELSE
                                F_RAMP_pump:=1500; R_RAMP_pump:=TO_INT(PAR_NegFull_y);
                                IF  PWM_JOYY_L_UP>10 THEN
                                 F_RAMP_pump:=1500; R_RAMP_pump:=300;
                                END_IF
                        END_IF                
                4:
                        IF MainWinch_move AND (JiaYa_move OR CANO_JiayaPressure>80)  THEN
                                F_RAMP_pump:=1500; R_RAMP_pump:=150;
                        ELSE
                                F_RAMP_pump:=1500; R_RAMP_pump:=TO_INT(PAR_PosFull_y);//从200降
                                IF  PWM_JOYY_L_UP>10 THEN
                                 F_RAMP_pump:=1500; R_RAMP_pump:=300;
                                END_IF
                        END_IF                                
                5:
                        IF MainWinch_move AND (JiaYa_move OR CANO_JiayaPressure>80)  THEN
                                F_RAMP_pump:=1500; R_RAMP_pump:=200;
                        ELSE
                                F_RAMP_pump:=1500; R_RAMP_pump:=TO_INT(PAR_Zero_y);
                                IF  PWM_JOYY_L_UP>10 THEN
                                 F_RAMP_pump:=1500; R_RAMP_pump:=300;
                                END_IF
                        END_IF                        
                6:		IF MainWinch_move AND (JiaYa_move OR CANO_JiayaPressure>80)  THEN
                                F_RAMP_pump:=1500; R_RAMP_pump:=200;
                        ELSE
                                F_RAMP_pump:=1500; R_RAMP_pump:=200;
                                IF  PWM_JOYY_L_UP>10 THEN
                                 F_RAMP_pump:=1500; R_RAMP_pump:=300;
                                END_IF
                        END_IF               
         END_CASE	
(*
	CASE AI_ECM2_Flag OF
		1:F_RAMP_pump:=1500; R_RAMP_pump:=100;		  
		2:F_RAMP_pump:=1500; R_RAMP_pump:=200;	
		3:
			IF MainWinch_move AND (JiaYa_move OR CANO_JiayaPressure>80)  THEN    //3泵同时起压时，降低主泵的加载速度，避免掉速熄火
				F_RAMP_pump:=1500; R_RAMP_pump:=150;
			ELSE
				F_RAMP_pump:=1500; R_RAMP_pump:=250;
			END_IF		
		4:
			IF MainWinch_move AND (JiaYa_move OR CANO_JiayaPressure>80)  THEN
				F_RAMP_pump:=1500; R_RAMP_pump:=180;
			ELSE
				F_RAMP_pump:=1500; R_RAMP_pump:=300;
			END_IF				
		5:
			IF MainWinch_move AND (JiaYa_move OR CANO_JiayaPressure>80)  THEN
				F_RAMP_pump:=1500; R_RAMP_pump:=250;
			ELSE
				F_RAMP_pump:=1500; R_RAMP_pump:=300;
			END_IF			
		6:F_RAMP_pump:=1500; R_RAMP_pump:=300;	
	END_CASE	
*)


(******斜坡增步长300 斜坡降步长400->1500*****)	
RAMP15(
	IN:=UINT_TO_INT(RAMP15_IN), 
	ASCEND:= R_RAMP_pump, 
	DESCEND:= F_RAMP_pump, 
	TIMEBASE:=T#1000MS , 
	RESET:=FALSE , 
	OUT=>(PWM_Y1_SET));
(******减斜坡300->400*****)	
RAMP16(
	IN:=UINT_TO_INT(RAMP16_IN), 
	ASCEND:= R_RAMP_pump, 
	DESCEND:= F_RAMP_pump, 
	TIMEBASE:=T#1000MS , 
	RESET:=FALSE , 
	OUT=>(PWM_Y2_SET));

	
IF (NOT Rotation_move) AND (NOT MainWinch_move) AND (NOT PowerHead_move)
		AND (NOT JiaYa_move) AND (NOT ViceWinch_move)
		AND (NOT LeftMove_move) AND (NOT RightMove_move)  THEN
	PWM_Y1_Target:=0;
	PWM_Y2_Target:=0;
END_IF


IF PWM_Y1_SET<TO_INT(PAR_Y1_1_NegFull )THEN
	PWM_Y1_SET:=TO_INT(PAR_Y1_1_NegFull);
END_IF

IF PWM_Y2_SET<TO_INT(PAR_Y1_1_NegFull )THEN
	PWM_Y2_SET:=TO_INT(PAR_Y1_1_NegFull);
END_IF

IF(PWM_Y1_SET>1000) THEN
	PWM_Y1_SET := 300;
END_IF

IF(PWM_Y2_SET>1000) THEN
	PWM_Y2_SET := 300;
END_IF	
 //Y8 9 7 10执行
	PWM_Y8_SET_Target:=REAL_TO_UINT(UINT_TO_REAL(PWM_JOYY_L_UP)/1000*(PAR_Valve1_PosFull-PAR_Valve1_NegFull)+PAR_Valve1_NegFull);
	PWM_Y10_SET_Target:=REAL_TO_UINT(UINT_TO_REAL(PWM_JOYY_L_UP)/1000*(PAR_Valve2_PosFull-PAR_Valve2_NegFull)+PAR_Valve2_NegFull);
	PWM_Y7_SET_Target:=0;
	PWM_Y9_SET_Target:=0;

 (*  //左手柄回收过程，Y8,Y10缓慢降			
	IF (JoyDesFlag) THEN
	PWM_Y8_SET_Target:=REAL_TO_UINT(INT_TO_REAL(PWM_JOYY_L_UP_1)/1000*(PAR_Valve1_PosFull-PAR_Valve1_NegFull)+PAR_Valve1_NegFull);
	PWM_Y10_SET_Target:=REAL_TO_UINT(INT_TO_REAL(PWM_JOYY_L_UP_1)/1000*(PAR_Valve2_PosFull-PAR_Valve2_NegFull)+PAR_Valve2_NegFull);
	END_IF
*)	
	//Y7 8 9 10处理	
	//主卷扬根据阀的开关调整斜坡值	
		IF(PWM_Y8_SET<1000  AND  PWM_Y8_SET>=900)THEN    //主卷下放斜坡值
				F_RAMP_mainwinch_down:=200;
			
			ELSIF(PWM_Y8_SET<900)THEN
				F_RAMP_mainwinch_down:=400;
			ELSE
				F_RAMP_mainwinch_down:=400;
			END_IF
			
		IF(PWM_Y7_SET<1000  AND  PWM_Y7_SET>=900)THEN  //主卷上提斜坡值
				F_RAMP_mainwinch_down:=300;
		ELSIF(PWM_Y7_SET<900  )THEN
				F_RAMP_mainwinch_down:=200;
		ELSE
				F_RAMP_mainwinch_down:=400;
		END_IF
			
	RAMP7(
		IN:=WORD_TO_INT(PWM_Y7_SET_Target), 
		ASCEND:= R_RAMP_mainwinch, 
		DESCEND:= F_RAMP_mainwinch_up, 
		TIMEBASE:=TIMEBASE_mainwinch , 
		RESET:=FALSE , 
		OUT=>(PWM_Y7_SET_Target1));
	IF(PWM_Y7_SET_Target1>=400) THEN
		Curve_input:=TO_UINT(PWM_Y7_SET_Target1 - 400);
		IF(Curve_input>900) THEN
			Curve_input:=900;
		END_IF
		curve7(input:=REAL_TO_UINT(UINT_TO_REAL(Curve_input)*72.8),Zero:=FALSE,Full:=FALSE,
			   PAR_Progression:=Curve_Par,OutputEnable:=TRUE);
		PWM_Y7_SET:=PAR_Valve1_NegFull + REAL_TO_UINT(UINT_TO_REAL(curve7.Output)/72.8);
	ELSE
		PWM_Y7_SET:=0;
	END_IF
	
	
	RAMP8(
		IN:=WORD_TO_INT(PWM_Y8_SET_Target), 
		ASCEND:= R_RAMP_mainwinch, 
		DESCEND:= F_RAMP_mainwinch_down, 
		TIMEBASE:=TIMEBASE_mainwinch , 
		RESET:=FALSE , 
		OUT=>(PWM_Y8_SET_Target1));
	IF(PWM_Y8_SET_Target1>=400) THEN
		Curve_input:=TO_UINT(PWM_Y8_SET_Target1 - 400);
		IF(Curve_input>900) THEN
			Curve_input:=900;
		END_IF
		curve8(input:=REAL_TO_UINT(UINT_TO_REAL(Curve_input)*72.8),Zero:=FALSE,Full:=FALSE,
			   PAR_Progression:=Curve_Par,OutputEnable:=TRUE);
		PWM_Y8_SET:=PAR_Valve1_NegFull + REAL_TO_UINT(UINT_TO_REAL(curve8.Output)/72.8);
	ELSE
		PWM_Y8_SET:=0;
	END_IF
	
	
	RAMP9(
		IN:=WORD_TO_INT(PWM_Y9_SET_Target), 
		ASCEND:= R_RAMP_mainwinch, 
		DESCEND:= F_RAMP_mainwinch_up, 
		TIMEBASE:=TIMEBASE_mainwinch , 
		RESET:=FALSE , 
		OUT=>(PWM_Y9_SET_Target1));
	IF(PWM_Y9_SET_Target1>=400) THEN
		Curve_input:=TO_UINT(PWM_Y9_SET_Target1 - 400);
		IF(Curve_input>900) THEN
			Curve_input:=900;
		END_IF
		curve9(input:=REAL_TO_UINT(UINT_TO_REAL(Curve_input)*72.8),Zero:=FALSE,Full:=FALSE,
			   PAR_Progression:=Curve_Par,OutputEnable:=TRUE);
		PWM_Y9_SET:=PAR_Valve1_NegFull + REAL_TO_UINT(UINT_TO_REAL(curve9.Output)/72.8);
	ELSE
		PWM_Y9_SET:=0;
	END_IF
	
	RAMP10(
		IN:=WORD_TO_INT(PWM_Y10_SET_Target), 
		ASCEND:= R_RAMP_mainwinch, 
		DESCEND:= F_RAMP_mainwinch_down, 
		TIMEBASE:=TIMEBASE_mainwinch , 
		RESET:=FALSE , 
		OUT=>(PWM_Y10_SET_Target1));
	IF(PWM_Y10_SET_Target1>=400) THEN
		Curve_input:=TO_UINT(PWM_Y10_SET_Target1 - 400);
		IF(Curve_input>900) THEN
			Curve_input:=900;
		END_IF
		curve10(input:=REAL_TO_UINT(UINT_TO_REAL(Curve_input)*72.8),Zero:=FALSE,Full:=FALSE,
			   PAR_Progression:=Curve_Par,OutputEnable:=TRUE);
		PWM_Y10_SET:=PAR_Valve1_NegFull + REAL_TO_UINT(UINT_TO_REAL(curve10.Output)/72.8);
	ELSE
		PWM_Y10_SET:=0;
	END_IF
  //Y7 8 9 10范围限制
	IF(PWM_Y7_SET>1300)THEN
		PWM_Y7_SET :=1300;
	END_IF
	IF(PWM_Y8_SET>1300)THEN
		PWM_Y8_SET :=1300;
	END_IF
	IF(PWM_Y9_SET>1300)THEN
		PWM_Y9_SET :=1300;
	END_IF
	IF(PWM_Y10_SET>1300)THEN
		PWM_Y10_SET :=1300;
	END_IF
	
	IF(PWM_Y7_SET<=300)THEN
		PWM_Y7_SET :=0;
	END_IF
	IF(PWM_Y8_SET<=300)THEN
		PWM_Y8_SET :=0;
	END_IF
	IF(PWM_Y9_SET<=300)THEN
		PWM_Y9_SET :=0;
	END_IF
	IF(PWM_Y10_SET<=300)THEN
		PWM_Y10_SET :=0;
	END_IF
	
//去除Y7Y9干扰
PWM_Y7_SET:=0;
PWM_Y9_SET:=0;
	
  //Y39 40执行
	(*主泵卸荷阀控制*)
		PWM_Y39_SET_Target:=MAX(PWM_Y8_SET_Target,PWM_Y7_SET_Target);
		PWM_Y40_SET_Target:=MAX(PWM_Y9_SET_Target,PWM_Y10_SET_Target);
	(*卸荷动作缓冲*)
(*RAMP19(
	IN:=WORD_TO_INT(PWM_Y39_SET_Target), 
	ASCEND:= R_RAMP_xiehe, 
	DESCEND:= F_RAMP_xiehe, 
	TIMEBASE:=TIMEBASE_xiehe , 
	RESET:=FALSE , 
	OUT=>(PWM_Y39_SET_Target1));
	*)
IF(PWM_Y39_SET_Target>=400) THEN
	Curve_input:=TO_UINT(PWM_Y39_SET_Target - 400);
	IF(Curve_input>900) THEN
		Curve_input:=900;
	END_IF
	curve19(input:=REAL_TO_UINT(UINT_TO_REAL(Curve_input)*72.8),Zero:=FALSE,Full:=FALSE,
		   PAR_Progression:=Curve_Par1,OutputEnable:=TRUE);
	PWM_Y39_SET:=PAR_Valve1_NegFull + REAL_TO_UINT(UINT_TO_REAL(curve19.Output)/72.8);
ELSE
	PWM_Y39_SET:=0;
END_IF

(*
RAMP20(
	IN:=WORD_TO_INT(PWM_Y40_SET_Target), 
	ASCEND:= R_RAMP_xiehe, 
	DESCEND:= F_RAMP_xiehe, 
	TIMEBASE:=TIMEBASE_xiehe , 
	RESET:=FALSE , 
	OUT=>(PWM_Y40_SET_Target1));
	*)
IF(PWM_Y40_SET_Target>=400) THEN
	Curve_input:=TO_UINT(PWM_Y40_SET_Target - 400);
	IF(Curve_input>900) THEN
		Curve_input:=900;
	END_IF
	curve20(input:=REAL_TO_UINT(UINT_TO_REAL(Curve_input)*72.8),Zero:=FALSE,Full:=FALSE,
		   PAR_Progression:=Curve_Par1,OutputEnable:=TRUE);
	PWM_Y40_SET:=PAR_Valve1_NegFull + REAL_TO_UINT(UINT_TO_REAL(curve20.Output)/72.8);
ELSE
	PWM_Y40_SET:=0;
END_IF
	
IF(PWM_Y39_SET>1300)THEN
	PWM_Y39_SET :=1300;
END_IF
IF(PWM_Y40_SET>1300)THEN
	PWM_Y40_SET :=1300;
END_IF

IF(PWM_Y39_SET<=300)THEN
	PWM_Y39_SET :=0;
END_IF
IF(PWM_Y40_SET<=300)THEN
	PWM_Y40_SET :=0;
END_IF

IF JiaYa_move THEN
	IF PWM_JOYY_R_UP>10 THEN//加压下
		PWM_Y23_SET_Taget:=REAL_TO_UINT(UINT_TO_REAL(PWM_JOYY_R_UP)/1000*(800-PAR_Valve3_NegFull)+PAR_Valve3_NegFull);
		PWM_Y24_SET_Taget:=0;
		
		IF(CANI_JiaYaFastSwitch OR DI_RHandle_SB7)THEN //加压快
			PWM_Y2_Target:=REAL_TO_UINT(UINT_TO_REAL(PWM_JOYY_R_UP)/1000*(500-300)+300);
			PWM_Y17_SET:=0;
			PWM_Y17_SET2:=0;
			PWM_Y18_SET_Taget:=1300;
		ELSE
			PWM_Y18_SET_Taget:=0;
		END_IF
		
	ELSIF PWM_JOYY_R_DOWN>10 THEN//加压上
		PWM_Y24_SET_Taget:=REAL_TO_UINT(UINT_TO_REAL(PWM_JOYY_R_DOWN)/1000*(800-PAR_Valve3_NegFull)+PAR_Valve3_NegFull);
		PWM_Y23_SET_Taget:=0;
		
		IF(CANI_JiaYaFastSwitch OR DI_RHandle_SB7)THEN //加压快
			PWM_Y2_Target:=REAL_TO_UINT(UINT_TO_REAL(PWM_JOYY_R_DOWN)/1000*(500-300)+300);
			PWM_Y17_SET:=800;
			PWM_Y17_SET2:=1300;
			PWM_Y18_SET:=0;
		ELSE
			PWM_Y18_SET:=0;
		END_IF
	END_IF
ELSE
	PWM_Y23_SET_Taget:=0;
	PWM_Y24_SET_Taget:=0;
	PWM_Y17_SET:=0;
	PWM_Y18_SET:=0;
	PWM_Y17_SET2:=0;
END_IF

RAMP22(
	IN:=WORD_TO_INT(PWM_Y23_SET_Taget), 
	ASCEND:= ASCEND_value, 
	DESCEND:= 5000, 
	TIMEBASE:=T#1000MS , 
	RESET:=FALSE , 
	OUT=>(PWM_Y23_SET_Taget1));
IF(PWM_Y23_SET_Taget1<310)THEN
		ASCEND_value:=6000;
ELSIF(PWM_Y23_SET_Taget1>=310 AND PWM_Y23_SET_Taget1<450)THEN
		ASCEND_value:=100;
ELSE
		ASCEND_value:=300;
END_IF
IF(PWM_Y23_SET_Taget1>=300) THEN
	Curve_input:=TO_UINT(PWM_Y23_SET_Taget1 - 300);
	IF(Curve_input>500) THEN
		Curve_input:=500;
	END_IF
	PWM_Y23_SET:=300 + Curve_input;
ELSE
	PWM_Y23_SET:=0;
END_IF

RAMP24(
	IN:=WORD_TO_INT(PWM_Y24_SET_Taget), 
	ASCEND:= 500, 
	DESCEND:= 500, 
	TIMEBASE:=T#300MS , 
	RESET:=FALSE , 
	OUT=>((PWM_Y24_SET)));
(*IF(PWM_Y24_SET_Taget1>=300) THEN
	Curve_input:=TO_UINT(PWM_Y24_SET_Taget1 - 300);
	IF(Curve_input>500) THEN
		Curve_input:=500;
	END_IF
	PWM_Y24_SET:=300 + Curve_input;
ELSE
	PWM_Y24_SET:=0;
END_IF*)



RAMP23(
	IN:=WORD_TO_INT(PWM_Y18_SET_Taget), 
	ASCEND:= ASCEND_value2, 
	DESCEND:= 5000, 
	TIMEBASE:=T#1000MS , 
	RESET:=FALSE , 
	OUT=>(PWM_Y18_SET_Taget1));
IF(PWM_Y18_SET_Taget1<610)THEN
		ASCEND_value2:=6000;
ELSE
	ASCEND_value2:=150;
END_IF	

IF(PWM_Y18_SET_Taget1>=600) THEN
	Curve_input:=TO_UINT(PWM_Y18_SET_Taget1 - 600);
	IF(Curve_input>700) THEN
		Curve_input:=700;
	END_IF
	PWM_Y18_SET:=600 + Curve_input;
ELSE
	PWM_Y18_SET:=0;
END_IF

(*PWM_Y23_SET:=PWM_Y23_SET_Taget;*)
IF JiaYa_move THEN
	IF PWM_JOYY_R_DOWN>10 THEN
		PWM_Y23_SET_Taget:=0;
		PWM_Y23_SET_Taget1:=0;
		PWM_Y23_SET:=0;
		PWM_Y18_SET_Taget1:=0;
		PWM_Y18_SET_Taget:=0;
		PWM_Y18_SET:=0;
	END_IF
END_IF

//加压限压
IF(CANI_DongLiTouPressLimitSwitch)THEN
	PWM_Y63_SET:=PAR_ValveD_PosFull;
ELSE
	PWM_Y63_SET:=0;
END_IF

END_PROGRAM

// StandardPLC/Application/SaveEngine/SaveEngineMode_2
PROGRAM SaveEngineMode_2
VAR
	EnergyEnable:BOOL;
	EnergyEnable1:BOOL;
	CasePWM_Y1:UINT;
	AcPre_w:REAL:=1;//蓄能器压力对应的主泵电流权重系数
	TON1:TON;
	Tension_Ton:TON;
	MainWinchTensionCase: UINT;
	Tension_Ton1: TON;
	Y39_TON:TON;
END_VAR



(*******************节能控制阀主阀主泵输出执行**************************)	
//ELSIF(GVL_SaveEngine.SaveEngineMode=2)THEN//节能上升模式	
	//2模式前500ms单泵工作，Y39为0，卸荷打开
	IF Mode2Timer>3 THEN
		PWM_Y39_SET_Target:=MAX(PWM_Y8_SET,PWM_Y7_SET_Target);
		RAMP19(
			IN:=WORD_TO_INT(PWM_Y39_SET_Target), 
			ASCEND:= R_RAMP_xiehe, 
			DESCEND:= F_RAMP_xiehe, 
			TIMEBASE:=TIMEBASE_xiehe , 
			RESET:=FALSE , 
			OUT=>(PWM_Y39_SET_Target1));
		IF(PWM_Y39_SET_Target1>=400) THEN
			Curve_input:=TO_UINT(PWM_Y39_SET_Target1 - 400);
		IF(Curve_input>900) THEN
			Curve_input:=900;
		END_IF
			curve19(input:=REAL_TO_UINT(UINT_TO_REAL(Curve_input)*72.8),Zero:=FALSE,Full:=FALSE,
		   PAR_Progression:=Curve_Par1,OutputEnable:=TRUE);
			PWM_Y39_SET:=PAR_Valve1_NegFull + REAL_TO_UINT(UINT_TO_REAL(curve19.Output)/72.8);
		ELSE
		 PWM_Y39_SET:=0;
		END_IF	
	ELSE
		PWM_Y39_SET:=0;
	END_IF

	GVL_SaveEngine.Y72OutPutState:=0;
	GVL_SaveEngine.Y71OutPutState:=1;
	
